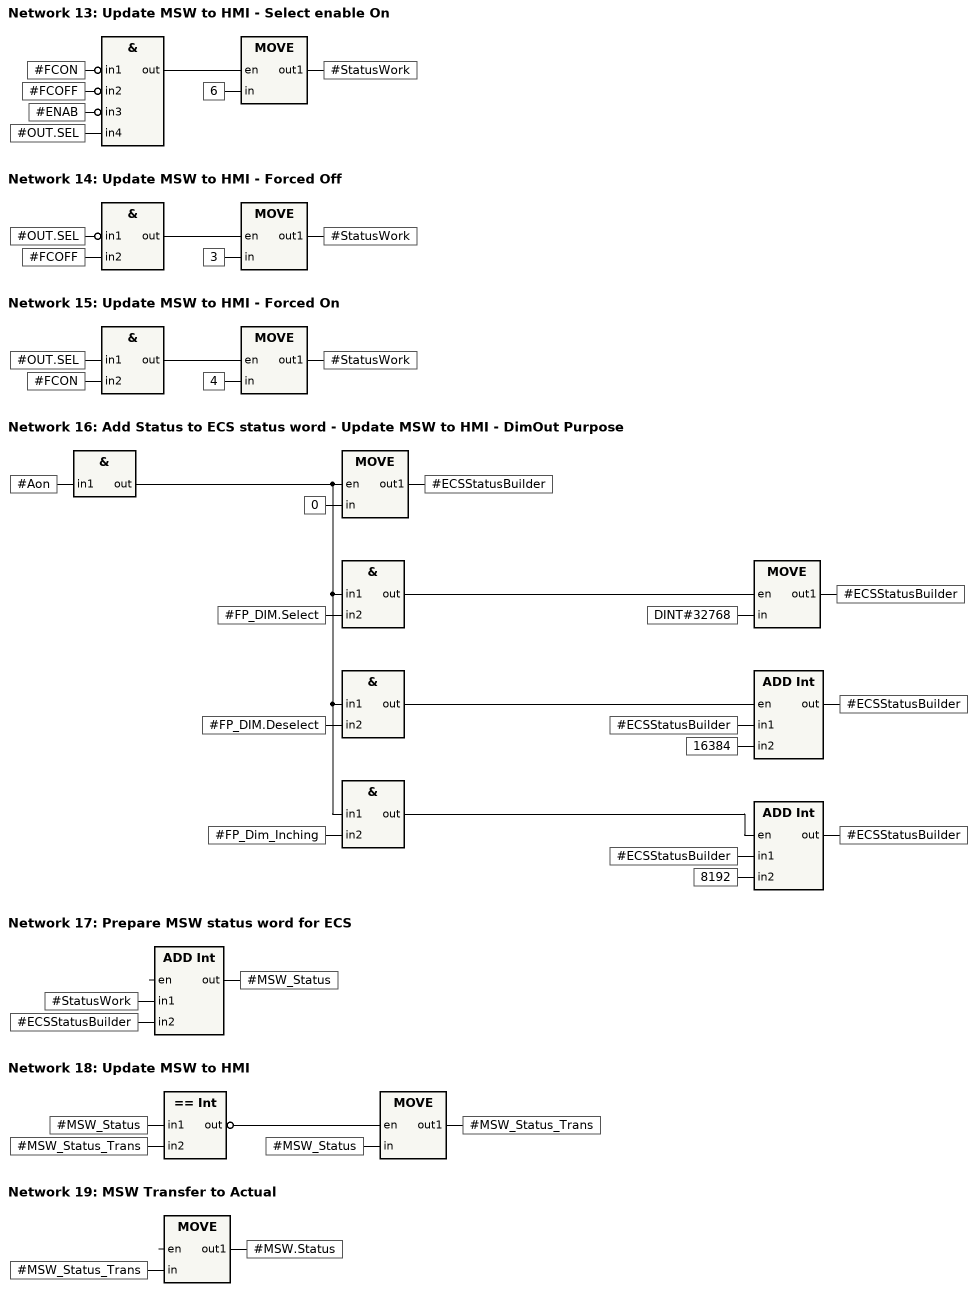
   IF NOT #FCON AND NOT #FCOFF AND NOT #ENAB AND #OUT.SEL THEN #StatusWork := 6; END_IF;
END_REGION

REGION Network 14: Update MSW to HMI - Forced Off
   IF NOT #OUT.SEL AND #FCOFF THEN #StatusWork := 3; END_IF;
END_REGION

REGION Network 15: Update MSW to HMI - Forced On
   IF #OUT.SEL AND #FCON THEN #StatusWork := 4; END_IF;
END_REGION

REGION Network 16: Add Status to ECS status word - Update MSW to HMI - DimOut Purpose
   // Bit 15 = 32768 - Dim_Select
   // Bit 14 = 16384 - Dim_Deselect
   // Bit 13 = 8192  - Dim Inching
   // Bit 12 = 4096 (spare)
   // Bit 11 = 2048 (spare)
   IF #Aon THEN #ECSStatusBuilder := 0; END_IF;
   IF #Aon AND #FP_DIM.Select THEN #ECSStatusBuilder := DINT#32768; END_IF;
   IF #Aon AND #FP_DIM.Deselect THEN #ECSStatusBuilder := #ECSStatusBuilder + 16384; END_IF;
   IF #Aon AND #FP_Dim_Inching THEN #ECSStatusBuilder := #ECSStatusBuilder + 8192; END_IF;
END_REGION

REGION Network 17: Prepare MSW status word for ECS
   #MSW_Status := #StatusWork + #ECSStatusBuilder;
END_REGION

REGION Network 18: Update MSW to HMI
   IF NOT (#MSW_Status = #MSW_Status_Trans) THEN #MSW_Status_Trans := #MSW_Status; END_IF;
END_REGION

REGION Network 19: MSW Transfer to Actual
   #MSW.Status := #MSW_Status_Trans;
END_REGION

REGION Network 20: Write STAT to OUT
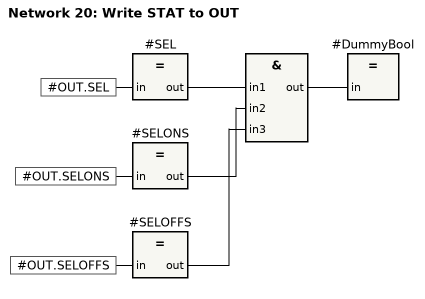
   #SEL := #OUT.SEL;
   #SELONS := #OUT.SELONS;
   #SELOFFS := #OUT.SELOFFS;
   #DummyBool := #OUT.SEL AND #OUT.SELONS AND #OUT.SELOFFS;
END_REGION
END_FUNCTION_BLOCK

FUNCTION_BLOCK "ACESYS_TOTALIZER"   // FB206, FBD
TITLE = ACESYS V8.0 - Build 002 - TOTALIZER
{ S7_Optimized_Access := 'FALSE' }
AUTHOR : FLSmidth
FAMILY : ACESYS
NAME : TOTALIZE
VERSION : 8.0
   VAR_INPUT
      CNT_EN : Bool;   // Counting Enable
      CNT : Bool;   // Counter Pulse
      RESET : Bool;   // Reset Counter Value
      DI_AI : Bool;   // Select Sum. Pulses or Analog-val ("0" = Dig./"1"=Ana.)
      AI : Real;   // Analog Value (Eng. Units)
   END_VAR
   VAR_OUTPUT
      COUNT : Real;   // Actual Counter Value
      Tot_Hour : Real;   // Tot. Totalizer, Base Hour
      Tot_Day : Real;   // Tot. Totalizer, Base Day
      Tot_Month : Real;
      Tot_Year : Real;   // Tot. Totalizer, Base Year
      MSW : DInt;
   END_VAR
   VAR_IN_OUT
      Token : "ACESYS_TOKEN";
   END_VAR
   VAR
      BlockInfo : Struct
         Ace_Version : Int;   // Acesys Block Version Number
         Ace_BuildNo : Int;   // Acesys Block Build Number
         State_Act : Int;   // Actual State Number
         State_Prev : Int;   // Previous State Number
         DB_Number : Int;   // Block Instance DB Number
      END_STRUCT;
      FP_CMD : Struct   // Faceplate Commands
         Spare_08 : Bool;
         Spare_09 : Bool;
         Spare_10 : Bool;
         Spare_11 : Bool;
         Spare_12 : Bool;
         Spare_13 : Bool;
         Spare_14 : Bool;
         AckAlarm : Bool;
         Reset : Bool;
         Spare_01 : Bool;
         Spare_02 : Bool;
         Spare_03 : Bool;
         Spare_04 : Bool;
         Spare_05 : Bool;
         Spare_06 : Bool;
         Spare_07 : Bool;
      END_STRUCT;
      FP_EN : Struct
         Reset : Bool;
      END_STRUCT;
      FP_SEL : Struct
         AI_Type_1 : Bool;   // Analog Value x/s
         AI_Type_2 : Bool;   // Analog Value x/min
         AI_Type_3 : Bool;   // Analog Value x/h
         COUNT_Factor_1 : Bool;   // AI / COUNT Ratio : 1:1
         COUNT_Factor_2 : Bool;   // AI / COUNT Ratio : 10:1
         COUNT_Factor_3 : Bool;   // AI / COUNT Ratio : 100:1
         COUNT_Factor_4 : Bool;   // AI / COUNT Ratio : 1000:1
         User_Hour : Bool;
         User_Day : Bool;
         User_Month : Bool;
         User_Year : Bool;
         User_Defined : Bool;
      END_STRUCT;
      FP_PAR : Struct
         Prev_Hour : Real;   // Save Old Counter register
         Prev_Day : Real;   // Save Old Counter register
         Prev_Month : Real;   // Save Old Counter register
         Prev_Year : Real;   // Save Old Counter register
         Prev_User : Real;   // Save Old Counter registe
      END_STRUCT;
      FP_DIM : Struct
         Reset : Bool;
      END_STRUCT;
      FP_SHOW : Struct
         Reset : Bool;
      END_STRUCT;
      ONS : Struct
         AI_Type_1 : Bool;
         AI_Type_2 : Bool;
         AI_Type_3 : Bool;
         COUNT_Factor_1 : Bool;
         COUNT_Factor_2 : Bool;
         COUNT_Factor_3 : Bool;
         COUNT_Factor_4 : Bool;
         User_Hour : Bool;
         User_Day : Bool;
         User_Month : Bool;
         User_Year : Bool;
         User_Defined : Bool;
         CNT : Bool;
         Reset : Bool;
         SecPulse1 : Bool;
         SecPulse2 : Bool;
      END_STRUCT;
      CMD_Reset : Bool;   // Reset Counters
      Sec_Pulse : Bool;
      Spare6 : Bool;
      Spare5 : Bool;
      Spare4 : Bool;
      Spare3 : Bool;
      Spare2 : Bool;
      Spare1 : Bool;
      inc_tmr_Real : LReal;   // Time elapsed since last block call (ms)
      IncrementVal : LReal;
      Selected_Factor : LReal;   // Ratio x:1
      Hour_Int : LReal;
      Day_Int : LReal;
      Month_Int : LReal;
      Year_Int : LReal;
      User_int : LReal;
      AI_Cal_Lreal : LReal;
      Runtime_RetVal : LReal;
      Runtime_Result : LReal;
      Runtime_Mem1 : LReal;
   END_VAR
   VAR_TEMP
      Aon : Bool;
      Aoff : Bool;
      DummyBool : Bool;
      DummyReal : Real;
      DummyLReal : LReal;
      DummyDint : DInt;
      AI_Cal : Real;
      DummyDword : DWord;
   END_VAR
   VAR_TEMP   // added for the SCL form of the ladder/FBD networks
      _w1 : Bool;
      _w2 : Bool;
   END_VAR
BEGIN

REGION Network 1
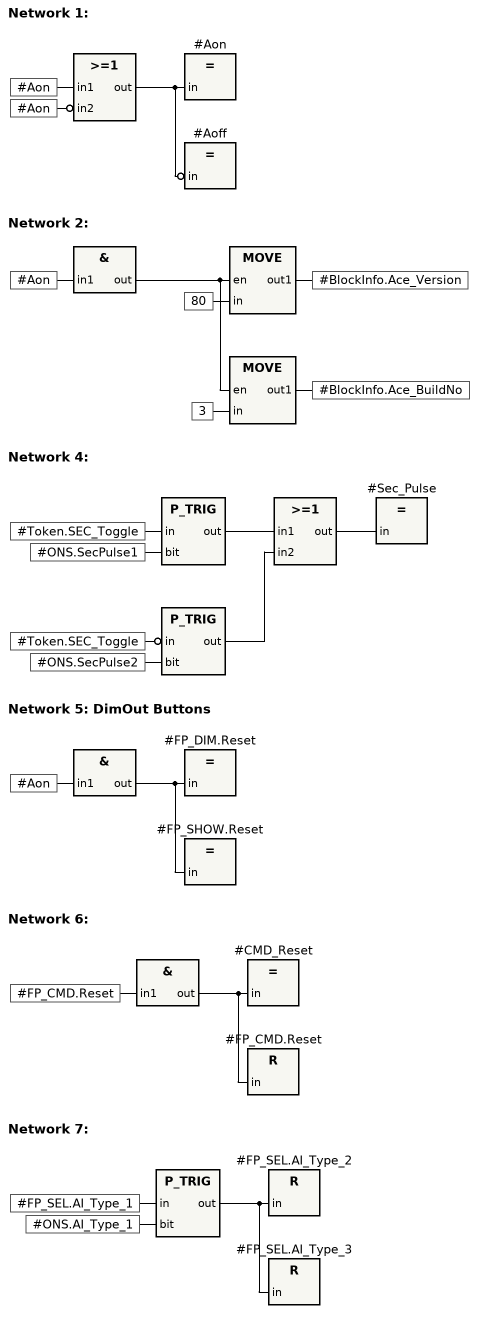
   #Aon := #Aon OR NOT #Aon;
   #Aoff := NOT #Aon;
END_REGION

REGION Network 2
   // Build 003 - Nw26 Runtime_Result replaced in Multiplication Input
   IF #Aon THEN
       #BlockInfo.Ace_Version := 80;
       #BlockInfo.Ace_BuildNo := 3;
   END_IF;
END_REGION

REGION Network 3 (STL): Instance DB Number to Faceplate
         L     DINO;
         T     #BlockInfo.DB_Number;
END_REGION

REGION Network 4
   #_w1 := #Token.SEC_Toggle AND NOT #ONS.SecPulse1;   // rising edge
   #ONS.SecPulse1 := #Token.SEC_Toggle;
   #_w2 := NOT #Token.SEC_Toggle AND NOT #ONS.SecPulse2;   // rising edge
   #ONS.SecPulse2 := NOT #Token.SEC_Toggle;
   #Sec_Pulse := #_w1 OR #_w2;
END_REGION

REGION Network 5: DimOut Buttons
   #FP_DIM.Reset := #Aon;
   #FP_SHOW.Reset := #Aon;
END_REGION

REGION Network 6
   // >>>>>Automatic Dep_CMD when use of block interface<<<<<<
   #CMD_Reset := #FP_CMD.Reset;
   IF #FP_CMD.Reset THEN #FP_CMD.Reset := FALSE; END_IF;
END_REGION

REGION Network 7
   // >>>>>Select Time Base for Input Engineering Value<<<<<<
   // (sec, minute, hour)
   #_w1 := #FP_SEL.AI_Type_1 AND NOT #ONS.AI_Type_1;   // rising edge
   #ONS.AI_Type_1 := #FP_SEL.AI_Type_1;
   IF #_w1 THEN
       #FP_SEL.AI_Type_2 := FALSE;
       #FP_SEL.AI_Type_3 := FALSE;
   END_IF;
END_REGION

REGION Network 8
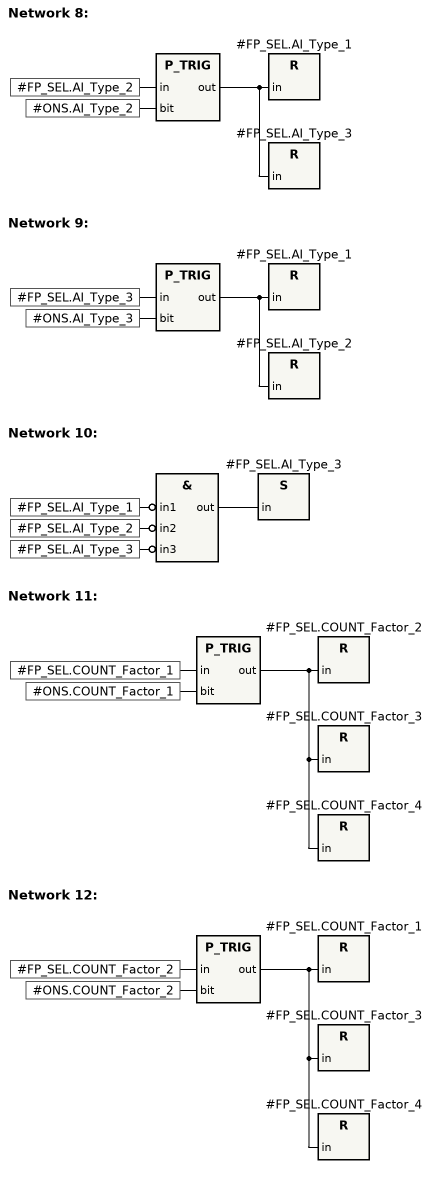
   #_w1 := #FP_SEL.AI_Type_2 AND NOT #ONS.AI_Type_2;   // rising edge
   #ONS.AI_Type_2 := #FP_SEL.AI_Type_2;
   IF #_w1 THEN
       #FP_SEL.AI_Type_1 := FALSE;
       #FP_SEL.AI_Type_3 := FALSE;
   END_IF;
END_REGION

REGION Network 9
   #_w1 := #FP_SEL.AI_Type_3 AND NOT #ONS.AI_Type_3;   // rising edge
   #ONS.AI_Type_3 := #FP_SEL.AI_Type_3;
   IF #_w1 THEN
       #FP_SEL.AI_Type_1 := FALSE;
       #FP_SEL.AI_Type_2 := FALSE;
   END_IF;
END_REGION

REGION Network 10
   IF NOT #FP_SEL.AI_Type_1 AND NOT #FP_SEL.AI_Type_2 AND NOT #FP_SEL.AI_Type_3 THEN
       #FP_SEL.AI_Type_3 := TRUE;
   END_IF;
END_REGION

REGION Network 11
   // >>>>>Select Factor<<<<<
   // (Ratio 1:1, 10:1, 100:1, 1000:1)
   #_w1 := #FP_SEL.COUNT_Factor_1 AND NOT #ONS.COUNT_Factor_1;   // rising edge
   #ONS.COUNT_Factor_1 := #FP_SEL.COUNT_Factor_1;
   IF #_w1 THEN
       #FP_SEL.COUNT_Factor_2 := FALSE;
       #FP_SEL.COUNT_Factor_3 := FALSE;
       #FP_SEL.COUNT_Factor_4 := FALSE;
   END_IF;
END_REGION

REGION Network 12
   #_w1 := #FP_SEL.COUNT_Factor_2 AND NOT #ONS.COUNT_Factor_2;   // rising edge
   #ONS.COUNT_Factor_2 := #FP_SEL.COUNT_Factor_2;
   IF #_w1 THEN
       #FP_SEL.COUNT_Factor_1 := FALSE;
       #FP_SEL.COUNT_Factor_3 := FALSE;
       #FP_SEL.COUNT_Factor_4 := FALSE;
   END_IF;
END_REGION

REGION Network 13
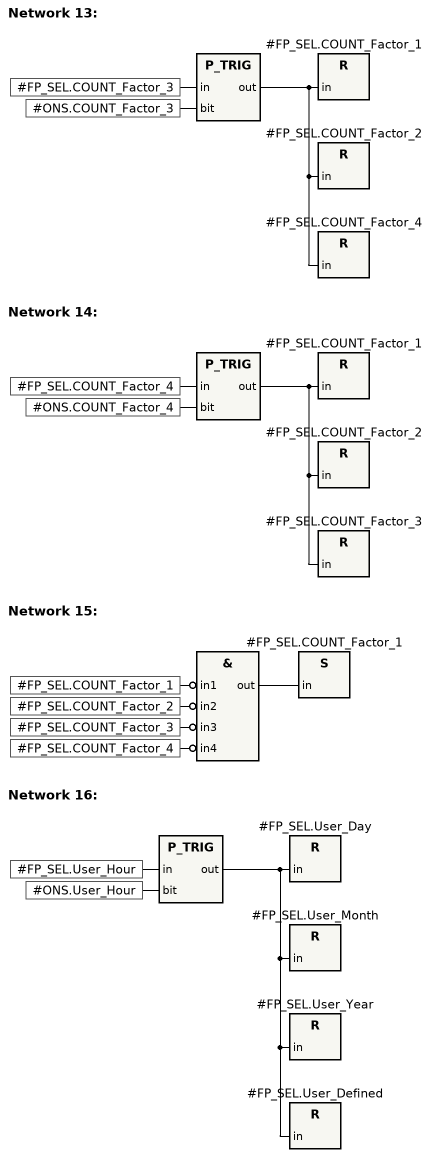
   #_w1 := #FP_SEL.COUNT_Factor_3 AND NOT #ONS.COUNT_Factor_3;   // rising edge
   #ONS.COUNT_Factor_3 := #FP_SEL.COUNT_Factor_3;
   IF #_w1 THEN
       #FP_SEL.COUNT_Factor_1 := FALSE;
       #FP_SEL.COUNT_Factor_2 := FALSE;
       #FP_SEL.COUNT_Factor_4 := FALSE;
   END_IF;
END_REGION

REGION Network 14
   #_w1 := #FP_SEL.COUNT_Factor_4 AND NOT #ONS.COUNT_Factor_4;   // rising edge
   #ONS.COUNT_Factor_4 := #FP_SEL.COUNT_Factor_4;
   IF #_w1 THEN
       #FP_SEL.COUNT_Factor_1 := FALSE;
       #FP_SEL.COUNT_Factor_2 := FALSE;
       #FP_SEL.COUNT_Factor_3 := FALSE;
   END_IF;
END_REGION

REGION Network 15
   IF NOT #FP_SEL.COUNT_Factor_1 AND NOT #FP_SEL.COUNT_Factor_2 AND NOT #FP_SEL.COUNT_Factor_3 AND NOT #FP_SEL.COUNT_Factor_4 THEN
       #FP_SEL.COUNT_Factor_1 := TRUE;
   END_IF;
END_REGION

REGION Network 16
   // >>>>>Select User Defined value to Output and  MSW<<<<<
   #_w1 := #FP_SEL.User_Hour AND NOT #ONS.User_Hour;   // rising edge
   #ONS.User_Hour := #FP_SEL.User_Hour;
   IF #_w1 THEN
       #FP_SEL.User_Day := FALSE;
       #FP_SEL.User_Month := FALSE;
       #FP_SEL.User_Year := FALSE;
       #FP_SEL.User_Defined := FALSE;
   END_IF;
END_REGION

REGION Network 17
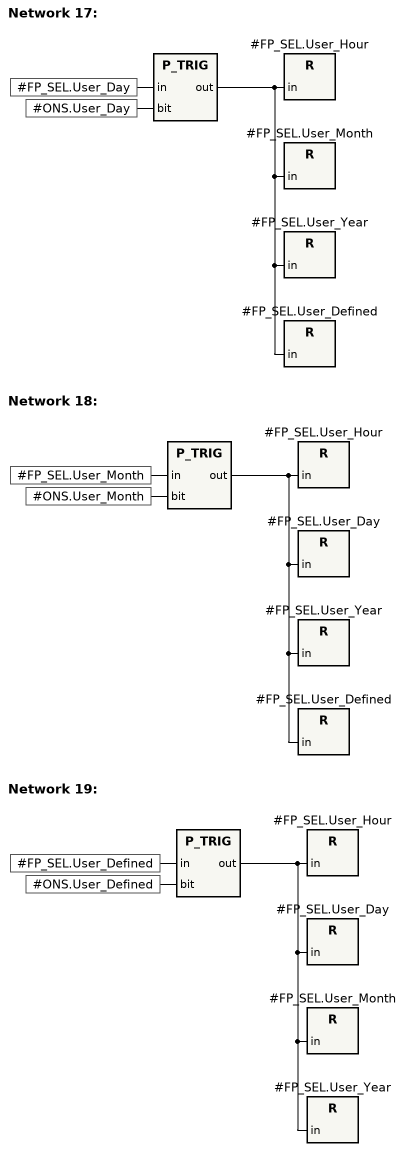
   #_w1 := #FP_SEL.User_Day AND NOT #ONS.User_Day;   // rising edge
   #ONS.User_Day := #FP_SEL.User_Day;
   IF #_w1 THEN
       #FP_SEL.User_Hour := FALSE;
       #FP_SEL.User_Month := FALSE;
       #FP_SEL.User_Year := FALSE;
       #FP_SEL.User_Defined := FALSE;
   END_IF;
END_REGION

REGION Network 18
   #_w1 := #FP_SEL.User_Month AND NOT #ONS.User_Month;   // rising edge
   #ONS.User_Month := #FP_SEL.User_Month;
   IF #_w1 THEN
       #FP_SEL.User_Hour := FALSE;
       #FP_SEL.User_Day := FALSE;
       #FP_SEL.User_Year := FALSE;
       #FP_SEL.User_Defined := FALSE;
   END_IF;
END_REGION

REGION Network 19
   #_w1 := #FP_SEL.User_Defined AND NOT #ONS.User_Defined;   // rising edge
   #ONS.User_Defined := #FP_SEL.User_Defined;
   IF #_w1 THEN
       #FP_SEL.User_Hour := FALSE;
       #FP_SEL.User_Day := FALSE;
       #FP_SEL.User_Month := FALSE;
       #FP_SEL.User_Year := FALSE;
   END_IF;
END_REGION

REGION Network 20
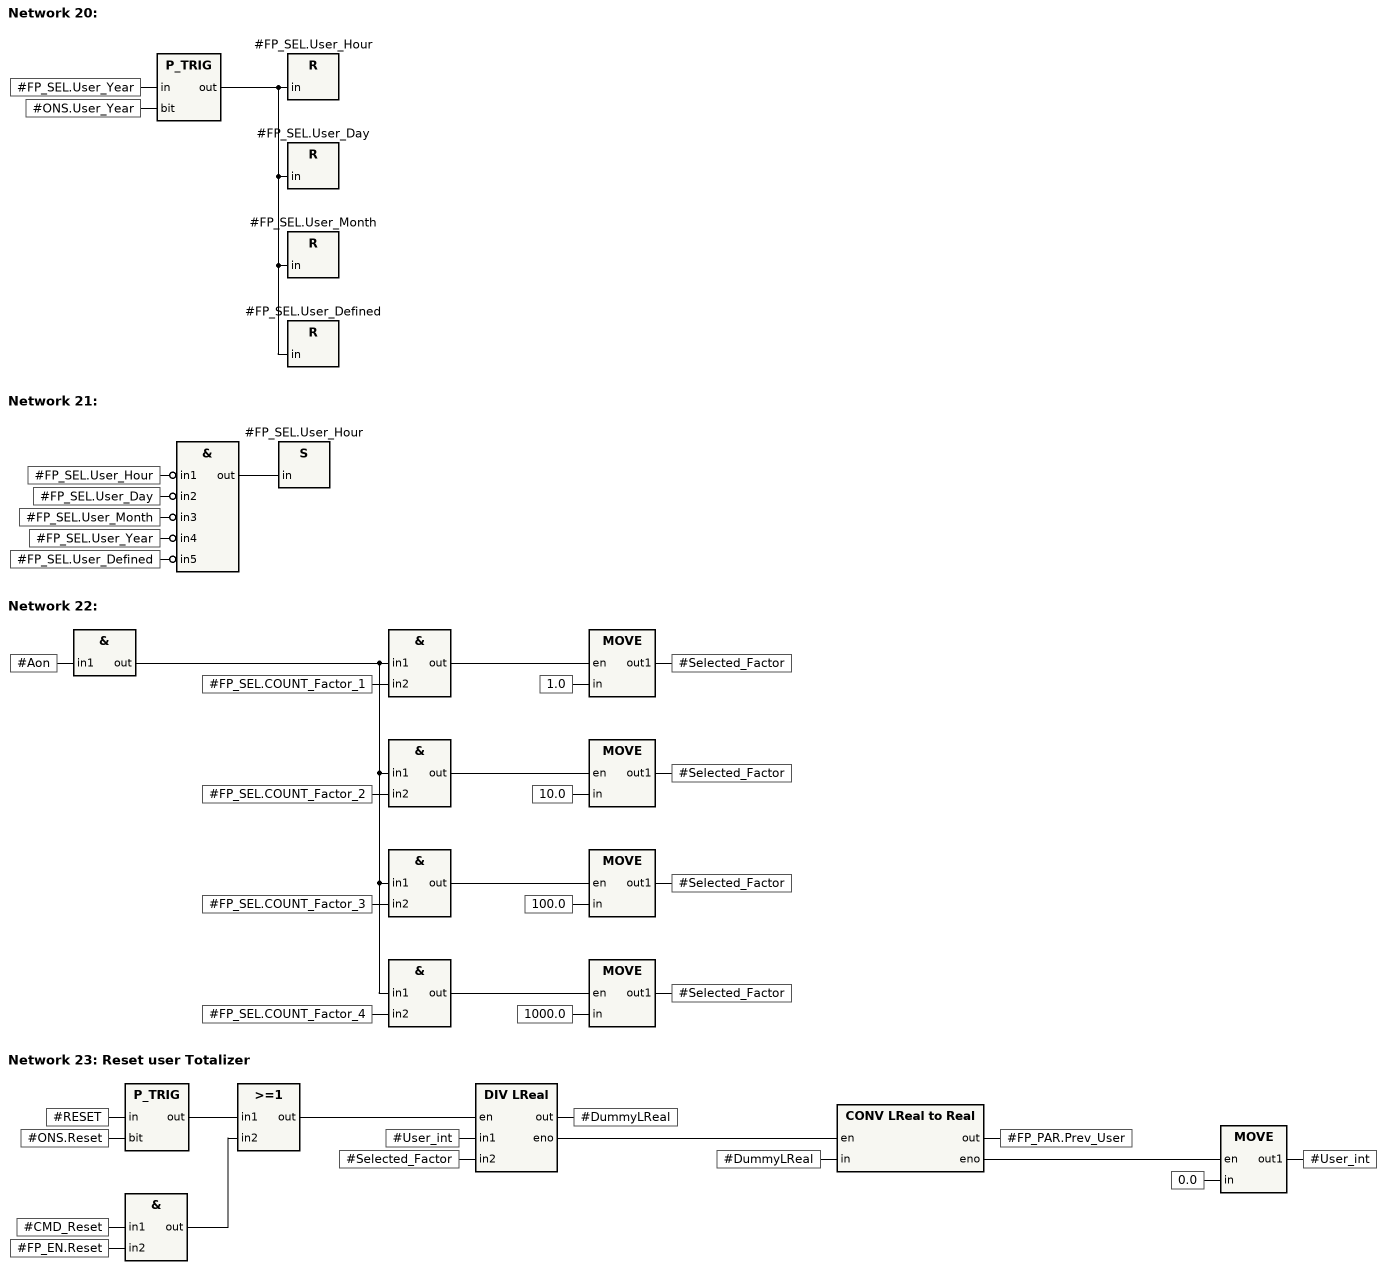
   #_w1 := #FP_SEL.User_Year AND NOT #ONS.User_Year;   // rising edge
   #ONS.User_Year := #FP_SEL.User_Year;
   IF #_w1 THEN
       #FP_SEL.User_Hour := FALSE;
       #FP_SEL.User_Day := FALSE;
       #FP_SEL.User_Month := FALSE;
       #FP_SEL.User_Defined := FALSE;
   END_IF;
END_REGION

REGION Network 21
   IF NOT #FP_SEL.User_Hour AND NOT #FP_SEL.User_Day AND NOT #FP_SEL.User_Month AND NOT #FP_SEL.User_Year AND NOT #FP_SEL.User_Defined THEN
       #FP_SEL.User_Hour := TRUE;
   END_IF;
END_REGION

REGION Network 22
   // >>>>>Get Selected Factor<<<<<
   IF #Aon AND #FP_SEL.COUNT_Factor_1 THEN #Selected_Factor := 1.0; END_IF;
   IF #Aon AND #FP_SEL.COUNT_Factor_2 THEN #Selected_Factor := 10.0; END_IF;
   IF #Aon AND #FP_SEL.COUNT_Factor_3 THEN #Selected_Factor := 100.0; END_IF;
   IF #Aon AND #FP_SEL.COUNT_Factor_4 THEN #Selected_Factor := 1000.0; END_IF;
END_REGION

REGION Network 23: Reset user Totalizer
   // Build 002 - 01.Feb.2016 : Factor is in included before the value is send to 
   // Prev_User
   // ENO of a box is taken as its EN; it also drops when the box reports an error
   #_w1 := #RESET AND NOT #ONS.Reset;   // rising edge
   #ONS.Reset := #RESET;
   IF #_w1 OR (#CMD_Reset AND #FP_EN.Reset) THEN
       #DummyLReal := #User_int / #Selected_Factor;
       #FP_PAR.Prev_User := LREAL_TO_REAL(#DummyLReal);
       #User_int := 0.0;
   END_IF;
END_REGION

REGION Network 24: Reset and Save prev. :Hour, Day, Month, Year
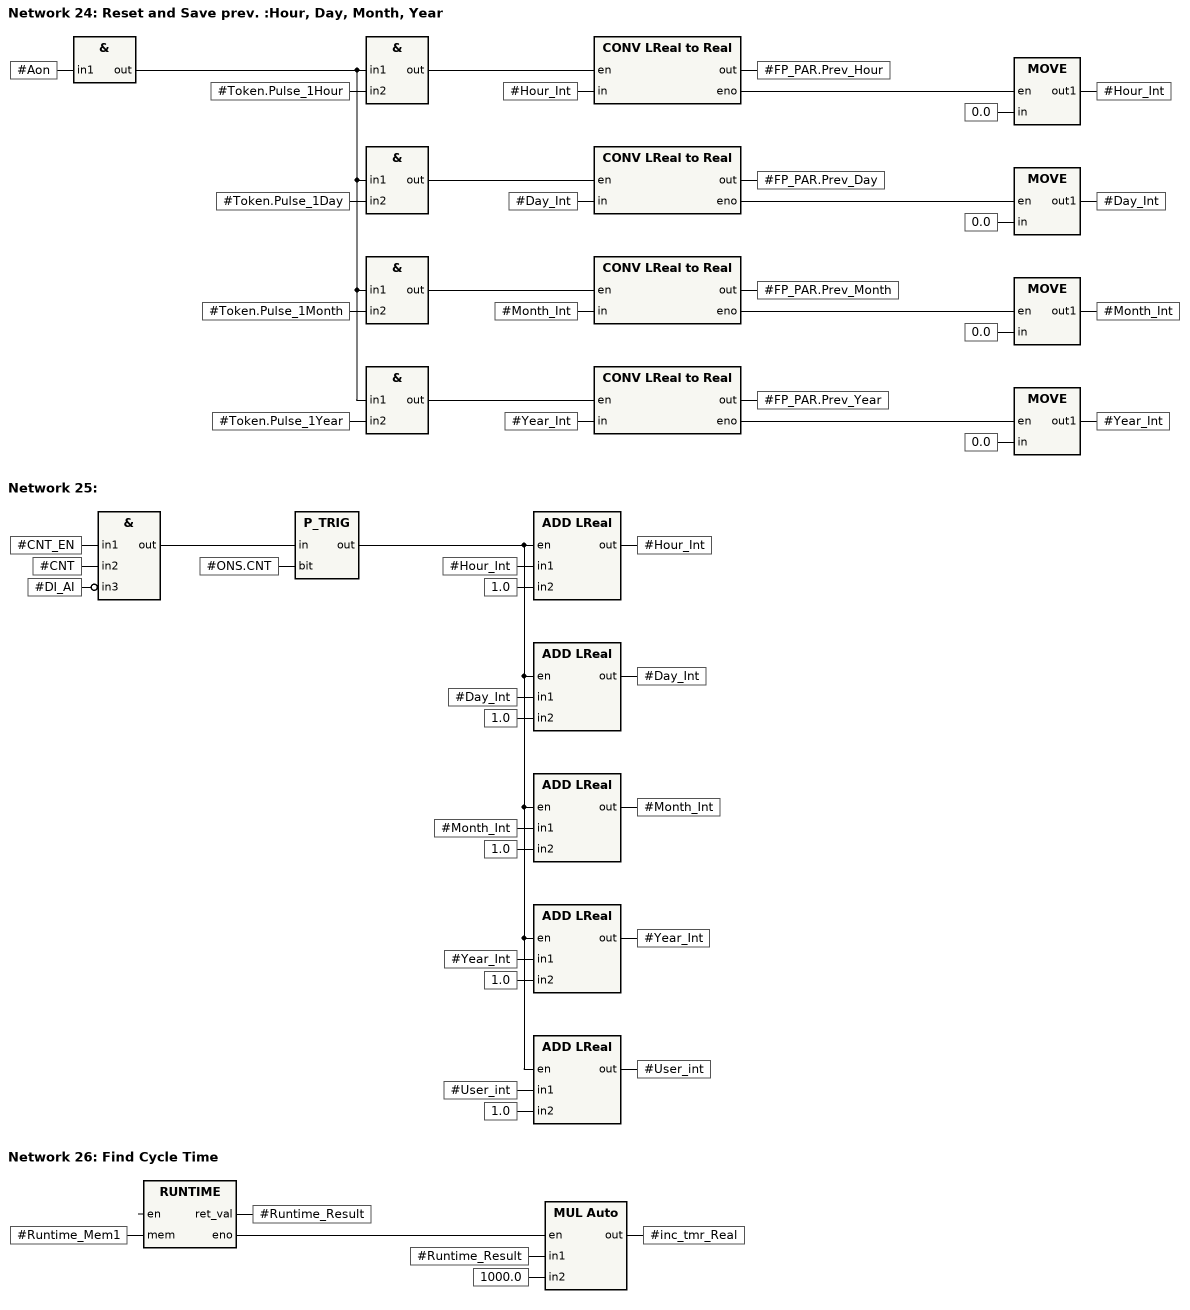
   IF #Aon AND #Token.Pulse_1Hour THEN
       #FP_PAR.Prev_Hour := LREAL_TO_REAL(#Hour_Int);
       #Hour_Int := 0.0;
   END_IF;
   IF #Aon AND #Token.Pulse_1Day THEN
       #FP_PAR.Prev_Day := LREAL_TO_REAL(#Day_Int);
       #Day_Int := 0.0;
   END_IF;
   IF #Aon AND #Token.Pulse_1Month THEN
       #FP_PAR.Prev_Month := LREAL_TO_REAL(#Month_Int);
       #Month_Int := 0.0;
   END_IF;
   IF #Aon AND #Token.Pulse_1Year THEN
       #FP_PAR.Prev_Year := LREAL_TO_REAL(#Year_Int);
       #Year_Int := 0.0;
   END_IF;
END_REGION

REGION Network 25
   // >>>>>Digital Counting<<<<<
   #_w1 := #CNT_EN AND #CNT AND NOT #DI_AI;
   #_w2 := #_w1 AND NOT #ONS.CNT;   // rising edge
   #ONS.CNT := #_w1;
   IF #_w2 THEN
       #Hour_Int := #Hour_Int + 1.0;
       #Day_Int := #Day_Int + 1.0;
       #Month_Int := #Month_Int + 1.0;
       #Year_Int := #Year_Int + 1.0;
       #User_int := #User_int + 1.0;
   END_IF;
END_REGION

REGION Network 26: Find Cycle Time
   // Build 003 - Runtime_Result replaced in Multiplication Input
   // no SCL statement known for Runtime: written as a call
   // ENO of a box is taken as its EN; it also drops when the box reports an error
   #Runtime_Result := Runtime(mem := #Runtime_Mem1);
   #inc_tmr_Real := #Runtime_Result * 1000.0;
END_REGION

REGION Network 27
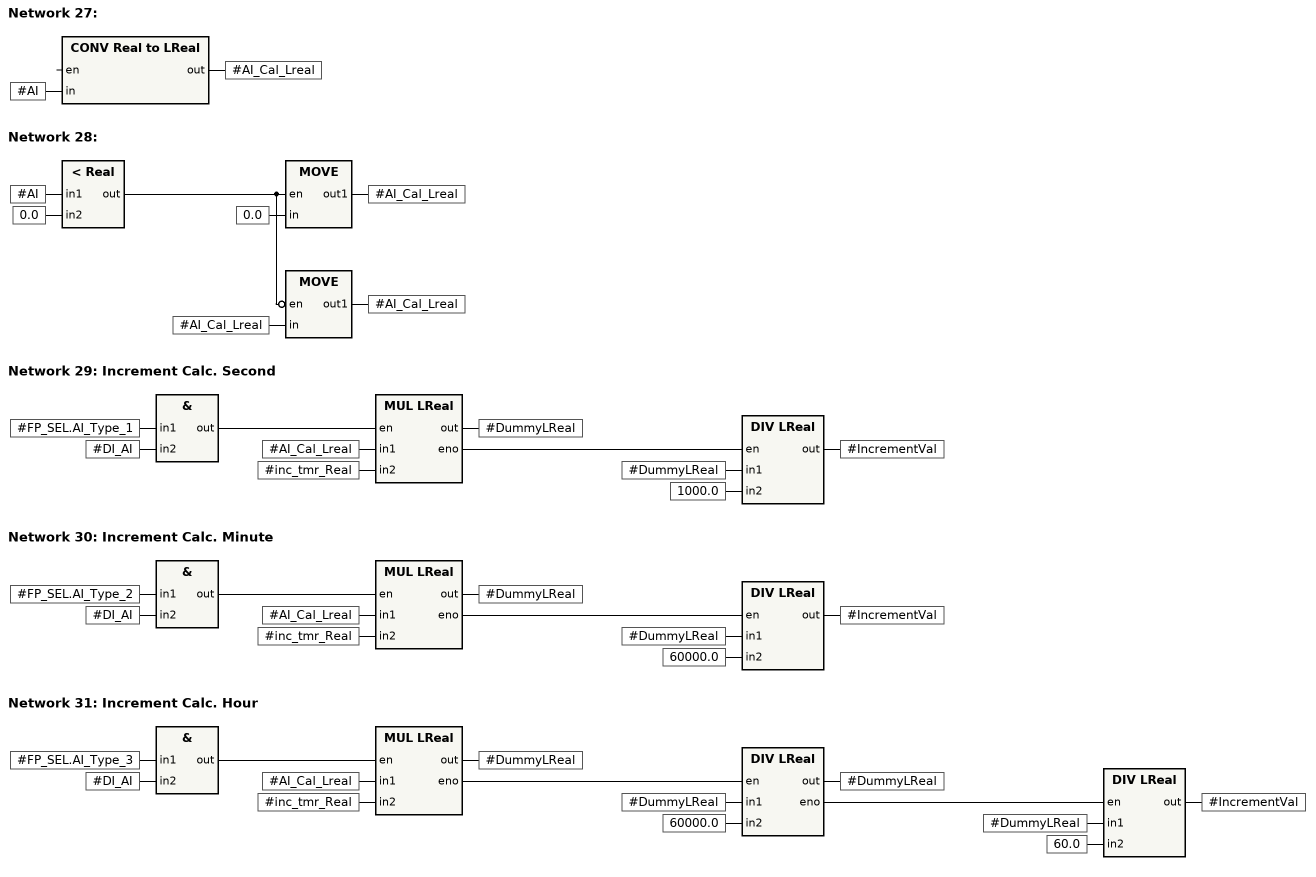
   #AI_Cal_Lreal := REAL_TO_LREAL(#AI);
END_REGION

REGION Network 28
   // Build 002 - 01.Feb.2016 : AI is clamped to "0"
   #_w1 := #AI < 0.0;
   IF #_w1 THEN #AI_Cal_Lreal := 0.0; END_IF;
   IF NOT #_w1 THEN #AI_Cal_Lreal := #AI_Cal_Lreal; END_IF;
END_REGION

REGION Network 29: Increment Calc. Second
   // Build 002 - 01.Feb.2016 : AI replaced with AI_Cal
   // ENO of a box is taken as its EN; it also drops when the box reports an error
   IF #FP_SEL.AI_Type_1 AND #DI_AI THEN
       #DummyLReal := #AI_Cal_Lreal * #inc_tmr_Real;
       #IncrementVal := #DummyLReal / 1000.0;
   END_IF;
END_REGION

REGION Network 30: Increment Calc. Minute
   // Build 002 - 01.Feb.2016 : AI replaced with AI_Cal
   // ENO of a box is taken as its EN; it also drops when the box reports an error
   IF #FP_SEL.AI_Type_2 AND #DI_AI THEN
       #DummyLReal := #AI_Cal_Lreal * #inc_tmr_Real;
       #IncrementVal := #DummyLReal / 60000.0;
   END_IF;
END_REGION

REGION Network 31: Increment Calc. Hour
   // Build 002 - 01.Feb.2016 : AI replaced with AI_Cal
   // ENO of a box is taken as its EN; it also drops when the box reports an error
   IF #FP_SEL.AI_Type_3 AND #DI_AI THEN
       #DummyLReal := #AI_Cal_Lreal * #inc_tmr_Real;
       #DummyLReal := #DummyLReal / 60000.0;
       #IncrementVal := #DummyLReal / 60.0;
   END_IF;
END_REGION

REGION Network 32
   // >>>>>Increment Base on Analog<<<<<
   // TOTAL Totalizer - Count up analog
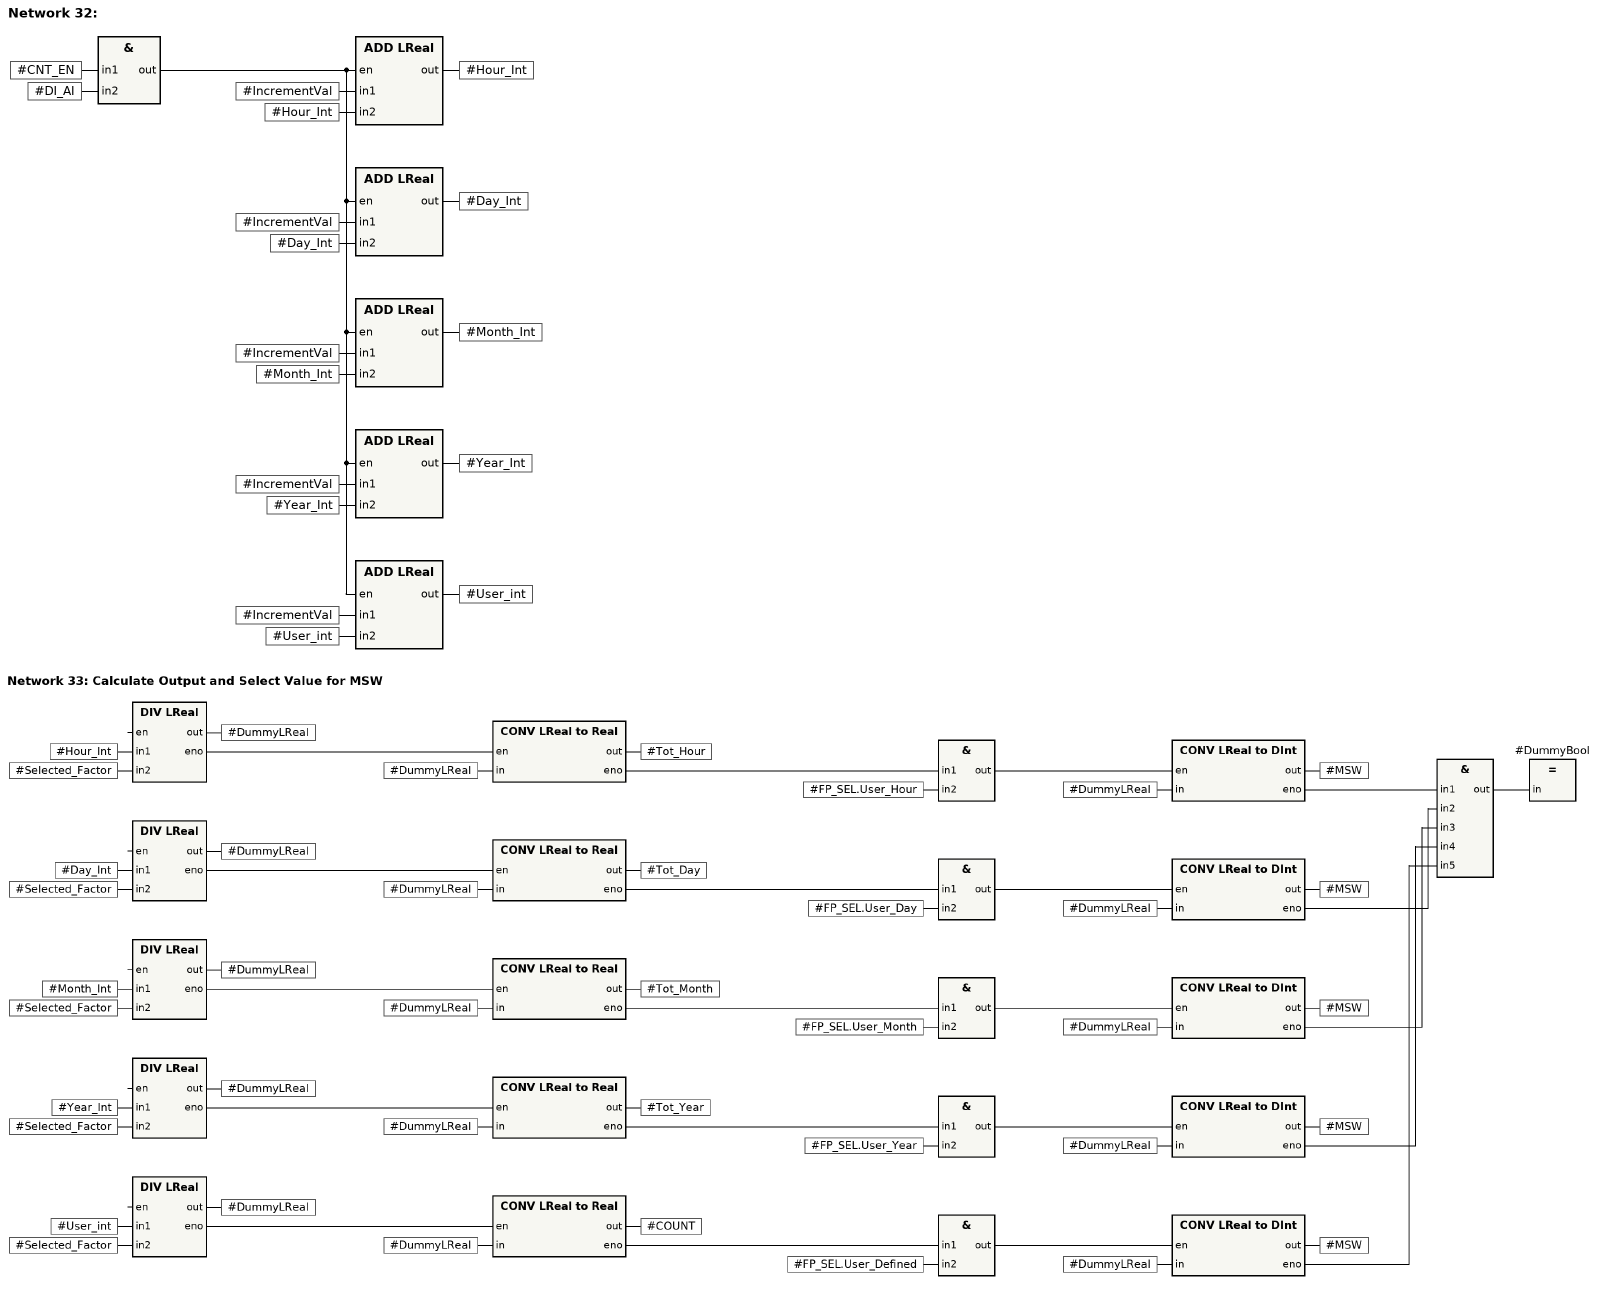
   IF #CNT_EN AND #DI_AI THEN
       #Hour_Int := #IncrementVal + #Hour_Int;
       #Day_Int := #IncrementVal + #Day_Int;
       #Month_Int := #IncrementVal + #Month_Int;
       #Year_Int := #IncrementVal + #Year_Int;
       #User_int := #IncrementVal + #User_int;
   END_IF;
END_REGION

REGION Network 33: Calculate Output and Select Value for MSW
   // ENO of a box is taken as its EN; it also drops when the box reports an error
   #DummyLReal := #Hour_Int / #Selected_Factor;
   #Tot_Hour := LREAL_TO_REAL(#DummyLReal);
   IF #FP_SEL.User_Hour THEN #MSW := LREAL_TO_DINT(#DummyLReal); END_IF;
   #DummyLReal := #Day_Int / #Selected_Factor;
   #Tot_Day := LREAL_TO_REAL(#DummyLReal);
   IF #FP_SEL.User_Day THEN #MSW := LREAL_TO_DINT(#DummyLReal); END_IF;
   #DummyLReal := #Month_Int / #Selected_Factor;
   #Tot_Month := LREAL_TO_REAL(#DummyLReal);
   IF #FP_SEL.User_Month THEN #MSW := LREAL_TO_DINT(#DummyLReal); END_IF;
   #DummyLReal := #Year_Int / #Selected_Factor;
   #Tot_Year := LREAL_TO_REAL(#DummyLReal);
   IF #FP_SEL.User_Year THEN #MSW := LREAL_TO_DINT(#DummyLReal); END_IF;
   #DummyLReal := #User_int / #Selected_Factor;
   #COUNT := LREAL_TO_REAL(#DummyLReal);
   IF #FP_SEL.User_Defined THEN #MSW := LREAL_TO_DINT(#DummyLReal); END_IF;
   #DummyBool := #FP_SEL.User_Hour AND #FP_SEL.User_Day AND #FP_SEL.User_Month AND #FP_SEL.User_Year AND #FP_SEL.User_Defined;
END_REGION
END_FUNCTION_BLOCK

FUNCTION_BLOCK "ACESYS_MD"   // FB207, FBD
TITLE = ACESYS V8.0 - Build 001 - MOTION DETECTOR
{ S7_Optimized_Access := 'FALSE' }
AUTHOR : FLSmidth
FAMILY : ACESYS
NAME : MotionDe
VERSION : 8.0
   VAR_INPUT
      CON : Bool;   // Start Command
      MD : Bool;   // Motion Signal
   END_VAR
   VAR_OUTPUT
      OK : Bool;   // Alarm Status OK
      MSW : "ACESYS_HMI_STAT_32T";
   END_VAR
   VAR_IN_OUT
      TOKEN : "ACESYS_TOKEN";
   END_VAR
   VAR
      BlockInfo : Struct
         Ace_Version : Int;   // Acesys Block Version Number
         Ace_BuildNo : Int;   // Acesys Block Build Number
         State_Act : Int;   // Actual State Number
         State_Prev : Int;   // Previous State Number
         DB_Number : Int;   // Block Instance DB Number
      END_STRUCT;
      FP_CMD : Struct   // Faceplate Commands
         Spare_08 : Bool;
         Spare_09 : Bool;
         Spare_10 : Bool;
         Spare_11 : Bool;
         Spare_12 : Bool;
         Spare_13 : Bool;
         Spare_14 : Bool;
         AckAlarm : Bool;
         Spare_00 : Bool;
         Spare_01 : Bool;
         Spare_02 : Bool;
         Spare_03 : Bool;
         Spare_04 : Bool;
         Spare_05 : Bool;
         Spare_06 : Bool;
         Spare_07 : Bool;
      END_STRUCT;
      FP_SEL : Struct
         MD_Maintain : Bool;
         MD_OnOff : Bool;
         MD_Puls : Bool;
         Keep_Status : Bool;
         MD_TimeBased : Bool;
      END_STRUCT;
      FP_PARM : Struct
         SpeedMonOffDelay_Acc : Int;
         SpeedMonOffDelay_Pre : Int;
         SpeedMonOnDelay_Acc : Int;
         SpeedMonOnDelay_Pre : Int;
         SpeedMonTrigDelay_Acc : Int;
         SpeedMonTrigDelay_Pre : Int;
         MD_Freq_SP : Int;
         MD_Freq_PV : Int;
         TimeBaseMonTime_Acc : Int;
         TimeBaseMonTime_Pre : Int;
         SpeedMonTimeBaseCNT_Acc : Int;
         SpeedMonTimeBaseCNT_Pre : Int;
      END_STRUCT;
      FP_EN : Struct
         ParentSupress : Bool;
      END_STRUCT;
      FP_SIM : "ACESYS_SIM_MD";
      ONS : Struct
         SecPulse1 : Bool;
         SecPulse2 : Bool;
         Acknowledge : Bool;
         MD_Pulse : Bool;
         MD_Maintain : Bool;
         MD_Type_OnOff : Bool;
         MD_Type_Pulse : Bool;
         MD_Type_TimeBased : Bool;
      END_STRUCT;
      StatusWork : Int;
      AlarmNo : Int;
      AlarmNo_Old : Int;
      Sec_Pulse : Bool;   // Pulse Every Second
      CMD_Acknowledge : Bool;
      ALARM_SuppresionActiv : Bool;
      ALARM_SuppresionActiv_1 : Bool;
      ALARM_AlarmPresent : Bool;
      ALARM_WarnPresent : Bool;
      ALARM_Failure_Ack_Requ : Bool;
      ALARM_Warn_Ack_Required : Bool;
      SpeedMonOnDelay_Done : Bool;
      SpeedMonOffDelay_Done : Bool;
      SpeedMonTrigDelay_Done : Bool;
      MD_Pulse : Bool;
      Keep_MD_Alarm : Bool;
      TimeBase_Done : Bool;
      TimeBase_TrigAlarm : Bool;
      SpeedMonOnDelay_Mem : Int;
      SpeedMonOffDelay_Mem : Int;
      SpeedMonTrigDelay_Mem : Int;
      TimeBaseMonTime_Mem : Int;
      MD_Time : DInt;
      MD_Time_DINT : DInt;
      MD_Timer : TON_TIME;
      OUT : Struct
         OK : Bool;
         MSW_EXT_ALARMFAILUNACK : Bool;
      END_STRUCT;
      MSW_Status_Trans : Int;
   END_VAR
   VAR_TEMP
      Aon : Bool;
      Aoff : Bool;
      DummyBool : Bool;
      DummyDInt : DInt;
   END_VAR
   VAR_TEMP   // added for the SCL form of the ladder/FBD networks
      _w1 : Bool;
      _w2 : Bool;
   END_VAR
BEGIN

REGION Network 1: Always On
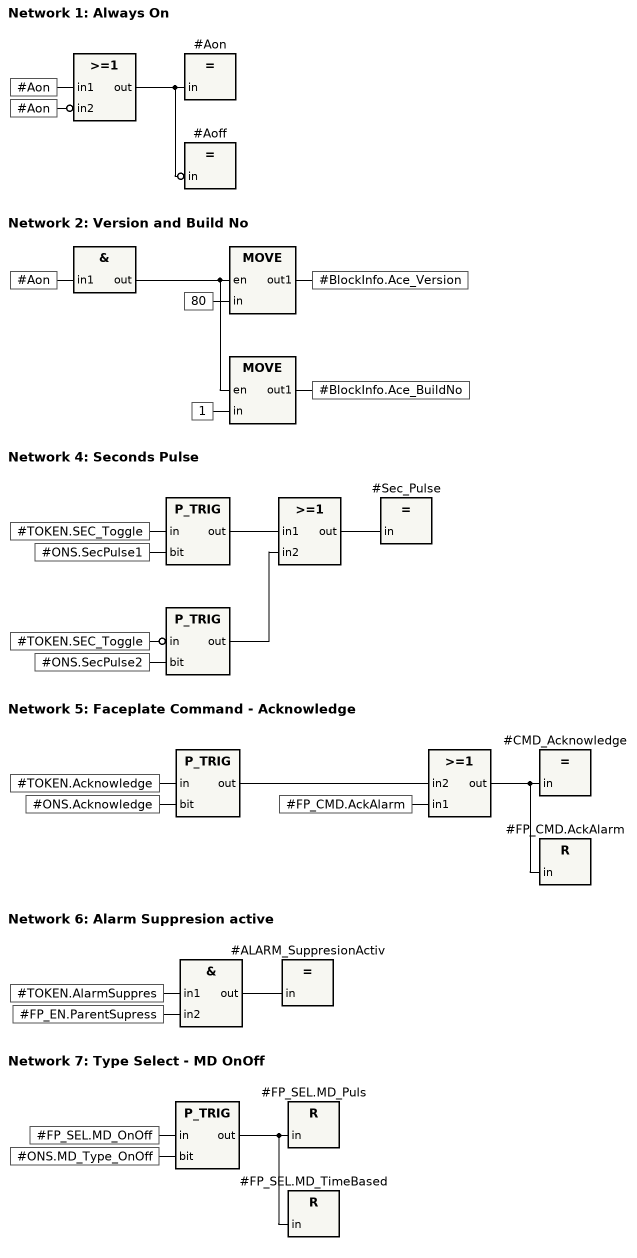
   #Aon := #Aon OR NOT #Aon;
   #Aoff := NOT #Aon;
END_REGION

REGION Network 2: Version and Build No
   IF #Aon THEN
       #BlockInfo.Ace_Version := 80;
       #BlockInfo.Ace_BuildNo := 1;
   END_IF;
END_REGION

REGION Network 3 (STL): Instance DB Number to Faceplate
         L     DINO;
         T     #BlockInfo.DB_Number;
END_REGION

REGION Network 4: Seconds Pulse
   #_w1 := #TOKEN.SEC_Toggle AND NOT #ONS.SecPulse1;   // rising edge
   #ONS.SecPulse1 := #TOKEN.SEC_Toggle;
   #_w2 := NOT #TOKEN.SEC_Toggle AND NOT #ONS.SecPulse2;   // rising edge
   #ONS.SecPulse2 := NOT #TOKEN.SEC_Toggle;
   #Sec_Pulse := #_w1 OR #_w2;
END_REGION

REGION Network 5: Faceplate Command - Acknowledge
   #_w1 := #TOKEN.Acknowledge AND NOT #ONS.Acknowledge;   // rising edge
   #ONS.Acknowledge := #TOKEN.Acknowledge;
   #CMD_Acknowledge := #_w1 OR #FP_CMD.AckAlarm;
   IF #CMD_Acknowledge THEN #FP_CMD.AckAlarm := FALSE; END_IF;
END_REGION

REGION Network 6: Alarm Suppresion active
   #ALARM_SuppresionActiv := #TOKEN.AlarmSuppres AND #FP_EN.ParentSupress;
END_REGION

REGION Network 7: Type Select - MD OnOff
   #_w1 := #FP_SEL.MD_OnOff AND NOT #ONS.MD_Type_OnOff;   // rising edge
   #ONS.MD_Type_OnOff := #FP_SEL.MD_OnOff;
   IF #_w1 THEN
       #FP_SEL.MD_Puls := FALSE;
       #FP_SEL.MD_TimeBased := FALSE;
   END_IF;
END_REGION

REGION Network 8: Type Select - MD Pulse
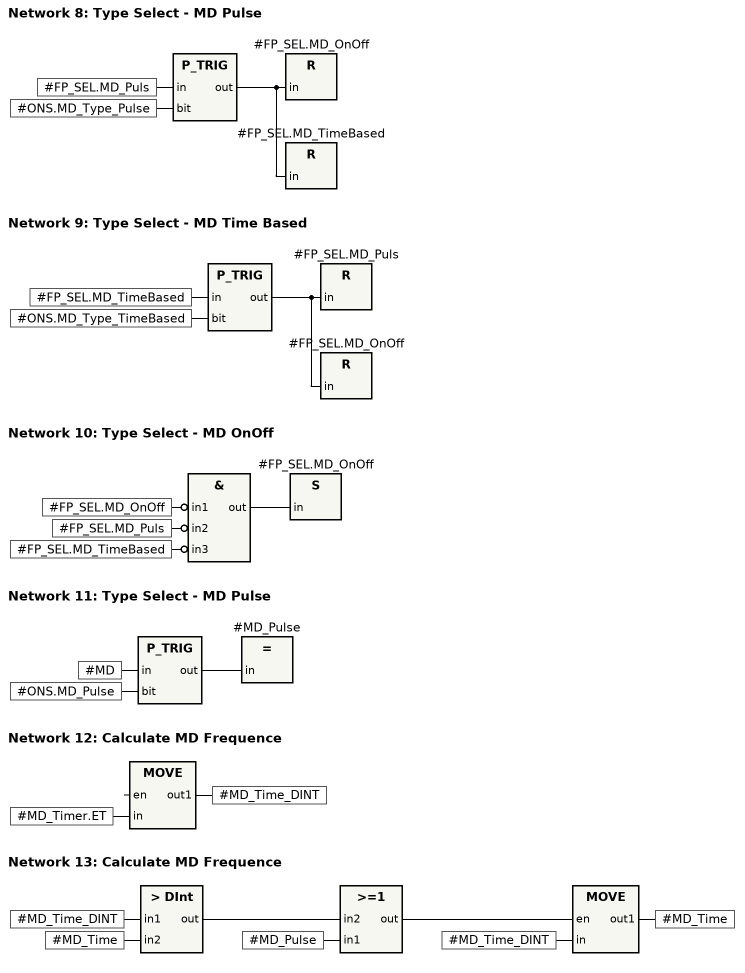
   #_w1 := #FP_SEL.MD_Puls AND NOT #ONS.MD_Type_Pulse;   // rising edge
   #ONS.MD_Type_Pulse := #FP_SEL.MD_Puls;
   IF #_w1 THEN
       #FP_SEL.MD_OnOff := FALSE;
       #FP_SEL.MD_TimeBased := FALSE;
   END_IF;
END_REGION

REGION Network 9: Type Select - MD Time Based
   #_w1 := #FP_SEL.MD_TimeBased AND NOT #ONS.MD_Type_TimeBased;   // rising edge
   #ONS.MD_Type_TimeBased := #FP_SEL.MD_TimeBased;
   IF #_w1 THEN
       #FP_SEL.MD_Puls := FALSE;
       #FP_SEL.MD_OnOff := FALSE;
   END_IF;
END_REGION

REGION Network 10: Type Select - MD OnOff
   IF NOT #FP_SEL.MD_OnOff AND NOT #FP_SEL.MD_Puls AND NOT #FP_SEL.MD_TimeBased THEN
       #FP_SEL.MD_OnOff := TRUE;
   END_IF;
END_REGION

REGION Network 11: Type Select - MD Pulse
   #_w1 := #MD AND NOT #ONS.MD_Pulse;   // rising edge
   #ONS.MD_Pulse := #MD;
   #MD_Pulse := #_w1;
END_REGION

REGION Network 12: Calculate MD Frequence
   #MD_Time_DINT := #MD_Timer.ET;
END_REGION

REGION Network 13: Calculate MD Frequence
   IF (#MD_Time_DINT > #MD_Time) OR #MD_Pulse THEN #MD_Time := #MD_Time_DINT; END_IF;
END_REGION

REGION Network 14: MD Timer
   // The MD_Timer is inserted twice to ensure that the timer is enabled in the same 
   // scan after af MD pulse.
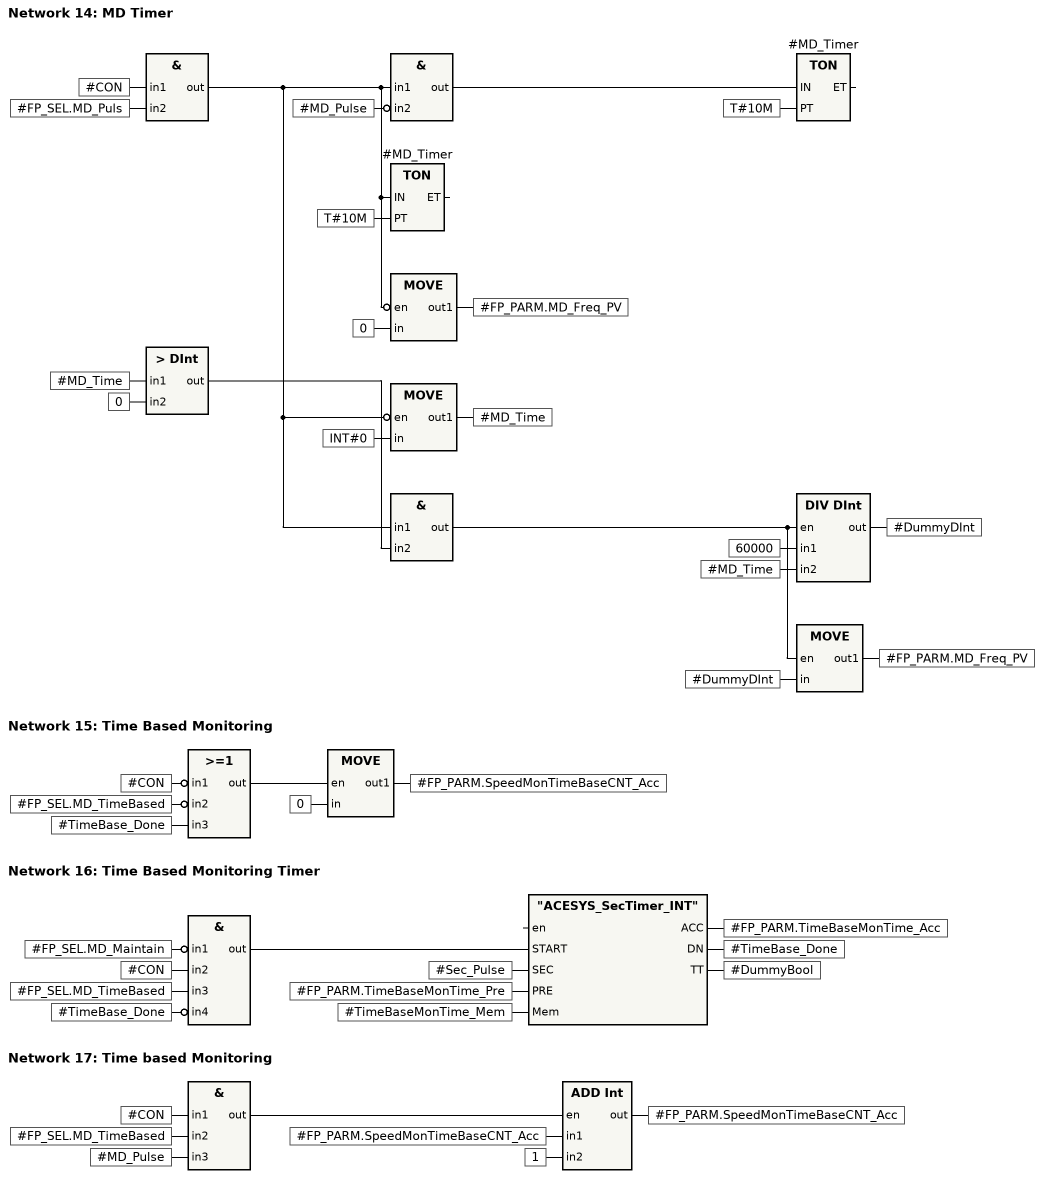
   #_w1 := #CON AND #FP_SEL.MD_Puls;
   #MD_Timer(IN := #_w1 AND NOT #MD_Pulse, PT := T#10M);   // TON
   #MD_Timer(IN := #_w1, PT := T#10M);   // TON
   IF NOT #_w1 THEN
       #FP_PARM.MD_Freq_PV := 0;
       #MD_Time := INT#0;
   END_IF;
   IF #_w1 AND (#MD_Time > 0) THEN
       #DummyDInt := 60000 / #MD_Time;
       #FP_PARM.MD_Freq_PV := #DummyDInt;
   END_IF;
END_REGION

REGION Network 15: Time Based Monitoring
   IF NOT #CON OR NOT #FP_SEL.MD_TimeBased OR #TimeBase_Done THEN
       #FP_PARM.SpeedMonTimeBaseCNT_Acc := 0;
   END_IF;
END_REGION

REGION Network 16: Time Based Monitoring Timer
   "ACESYS_SecTimer_INT"(START := NOT #FP_SEL.MD_Maintain AND #CON AND #FP_SEL.MD_TimeBased AND NOT #TimeBase_Done,
                         SEC := #Sec_Pulse,
                         PRE := #FP_PARM.TimeBaseMonTime_Pre,
                         Mem := #TimeBaseMonTime_Mem,
                         ACC => #FP_PARM.TimeBaseMonTime_Acc,
                         DN => #TimeBase_Done,
                         TT => #DummyBool);
END_REGION

REGION Network 17: Time based Monitoring
   IF #CON AND #FP_SEL.MD_TimeBased AND #MD_Pulse THEN
       #FP_PARM.SpeedMonTimeBaseCNT_Acc := #FP_PARM.SpeedMonTimeBaseCNT_Acc + 1;
   END_IF;
END_REGION

REGION Network 18: Time based Monitoring - Trig Alarm
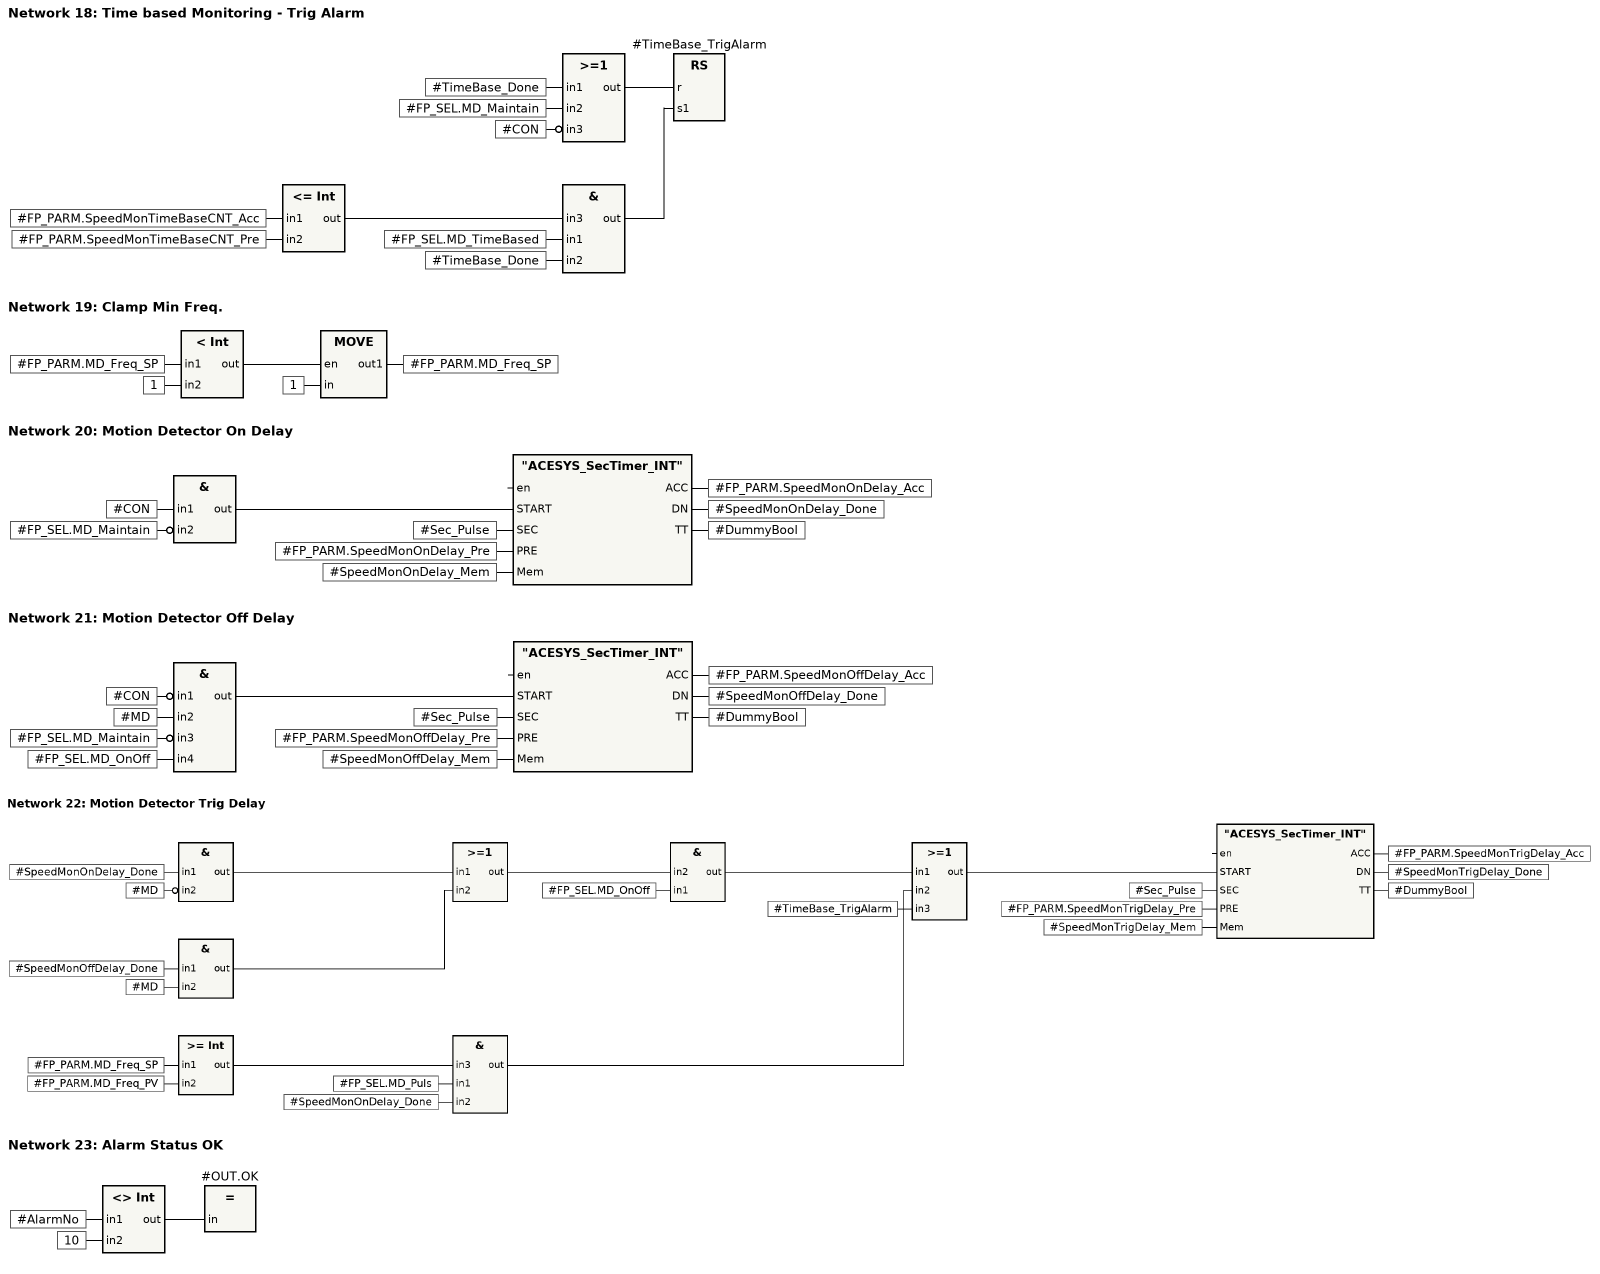
   IF #TimeBase_Done OR #FP_SEL.MD_Maintain OR NOT #CON THEN
       #TimeBase_TrigAlarm := FALSE;   // RS flip-flop
   END_IF;
   IF (#FP_PARM.SpeedMonTimeBaseCNT_Acc <= #FP_PARM.SpeedMonTimeBaseCNT_Pre) AND #FP_SEL.MD_TimeBased AND #TimeBase_Done THEN
       #TimeBase_TrigAlarm := TRUE;
   END_IF;
END_REGION

REGION Network 19: Clamp Min Freq.
   IF #FP_PARM.MD_Freq_SP < 1 THEN #FP_PARM.MD_Freq_SP := 1; END_IF;
END_REGION

REGION Network 20: Motion Detector On Delay
   "ACESYS_SecTimer_INT"(START := #CON AND NOT #FP_SEL.MD_Maintain,
                         SEC := #Sec_Pulse,
                         PRE := #FP_PARM.SpeedMonOnDelay_Pre,
                         Mem := #SpeedMonOnDelay_Mem,
                         ACC => #FP_PARM.SpeedMonOnDelay_Acc,
                         DN => #SpeedMonOnDelay_Done,
                         TT => #DummyBool);
END_REGION

REGION Network 21: Motion Detector Off Delay
   "ACESYS_SecTimer_INT"(START := NOT #CON AND #MD AND NOT #FP_SEL.MD_Maintain AND #FP_SEL.MD_OnOff,
                         SEC := #Sec_Pulse,
                         PRE := #FP_PARM.SpeedMonOffDelay_Pre,
                         Mem := #SpeedMonOffDelay_Mem,
                         ACC => #FP_PARM.SpeedMonOffDelay_Acc,
                         DN => #SpeedMonOffDelay_Done,
                         TT => #DummyBool);
END_REGION

REGION Network 22: Motion Detector Trig Delay
   "ACESYS_SecTimer_INT"(START := (((#SpeedMonOnDelay_Done AND NOT #MD) OR (#SpeedMonOffDelay_Done AND #MD)) AND #FP_SEL.MD_OnOff) OR ((#FP_PARM.MD_Freq_SP >= #FP_PARM.MD_Freq_PV) AND #FP_SEL.MD_Puls AND #SpeedMonOnDelay_Done) OR #TimeBase_TrigAlarm,
                         SEC := #Sec_Pulse,
                         PRE := #FP_PARM.SpeedMonTrigDelay_Pre,
                         Mem := #SpeedMonTrigDelay_Mem,
                         ACC => #FP_PARM.SpeedMonTrigDelay_Acc,
                         DN => #SpeedMonTrigDelay_Done,
                         TT => #DummyBool);
END_REGION

REGION Network 23: Alarm Status OK
   #OUT.OK := #AlarmNo <> 10;
END_REGION

REGION Network 24: Act as Dynamic sensor
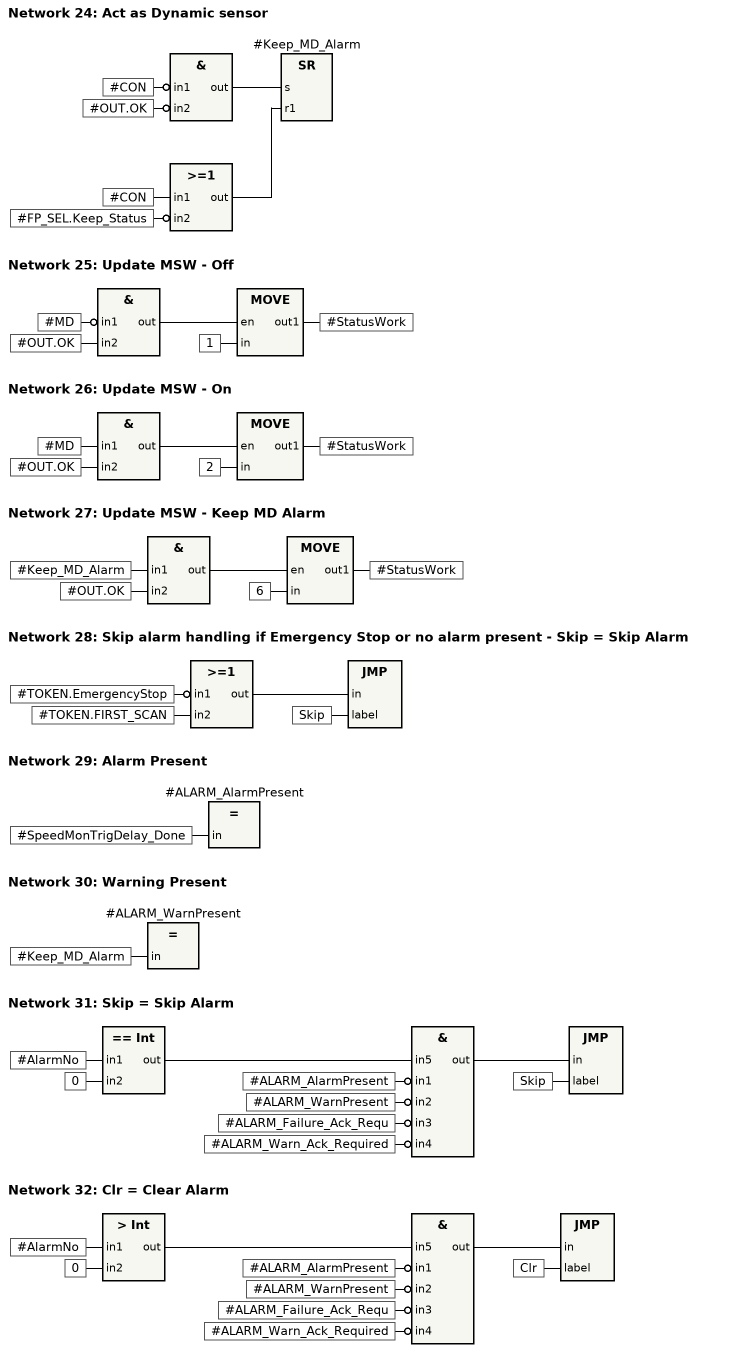
   IF NOT #CON AND NOT #OUT.OK THEN
       #Keep_MD_Alarm := TRUE;   // SR flip-flop
   END_IF;
   IF #CON OR NOT #FP_SEL.Keep_Status THEN #Keep_MD_Alarm := FALSE; END_IF;
END_REGION

REGION Network 25: Update MSW - Off
   IF NOT #MD AND #OUT.OK THEN #StatusWork := 1; END_IF;
END_REGION

REGION Network 26: Update MSW - On
   IF #MD AND #OUT.OK THEN #StatusWork := 2; END_IF;
END_REGION

REGION Network 27: Update MSW - Keep MD Alarm
   IF #Keep_MD_Alarm AND #OUT.OK THEN #StatusWork := 6; END_IF;
END_REGION

REGION Network 28: Skip alarm handling if Emergency Stop or no alarm present - Skip = Skip Alarm
   IF NOT #TOKEN.EmergencyStop OR #TOKEN.FIRST_SCAN THEN GOTO Skip; END_IF;
END_REGION

REGION Network 29: Alarm Present
   #ALARM_AlarmPresent := #SpeedMonTrigDelay_Done;
END_REGION

REGION Network 30: Warning Present
   #ALARM_WarnPresent := #Keep_MD_Alarm;
END_REGION

REGION Network 31: Skip = Skip Alarm
   IF (#AlarmNo = 0) AND NOT #ALARM_AlarmPresent AND NOT #ALARM_WarnPresent AND NOT #ALARM_Failure_Ack_Requ AND NOT #ALARM_Warn_Ack_Required THEN
       GOTO Skip;
   END_IF;
END_REGION

REGION Network 32: Clr = Clear Alarm
   IF (#AlarmNo > 0) AND NOT #ALARM_AlarmPresent AND NOT #ALARM_WarnPresent AND NOT #ALARM_Failure_Ack_Requ AND NOT #ALARM_Warn_Ack_Required THEN
       GOTO Clr;
   END_IF;
END_REGION

REGION Network 33: Ack = Alarm Acknowledge
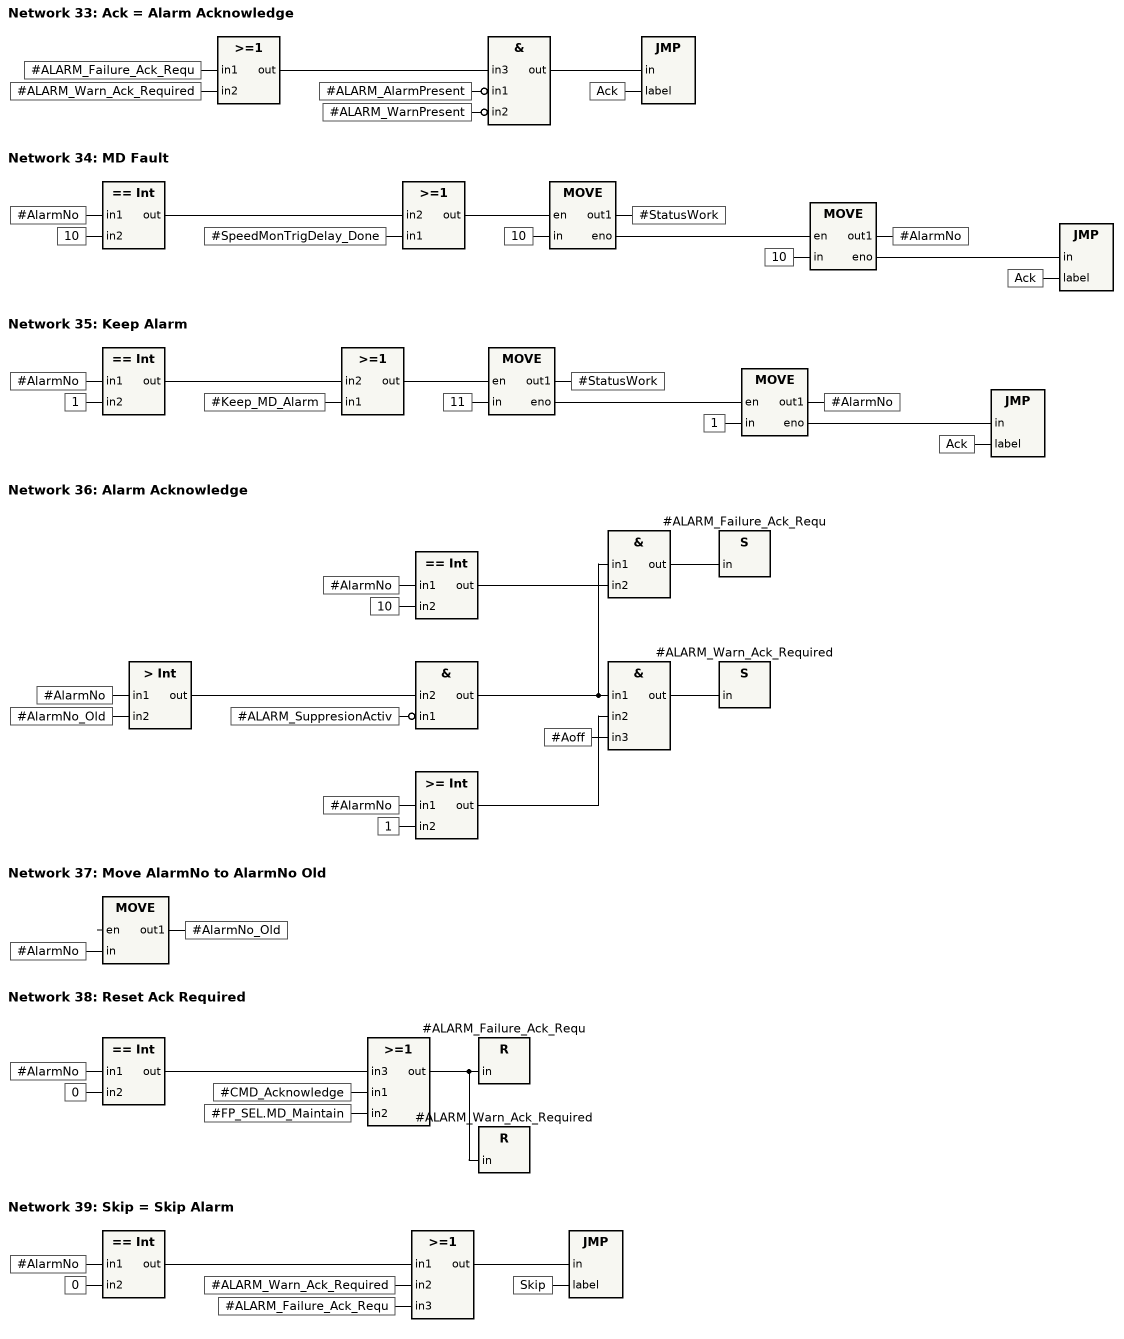
   IF (#ALARM_Failure_Ack_Requ OR #ALARM_Warn_Ack_Required) AND NOT #ALARM_AlarmPresent AND NOT #ALARM_WarnPresent THEN
       GOTO Ack;
   END_IF;
END_REGION

REGION Network 34: MD Fault
   // ENO of a box is taken as its EN; it also drops when the box reports an error
   #_w1 := (#AlarmNo = 10) OR #SpeedMonTrigDelay_Done;
   IF #_w1 THEN
       #StatusWork := 10;
       #AlarmNo := 10;
       GOTO Ack;
   END_IF;
END_REGION

REGION Network 35: Keep Alarm
   // ENO of a box is taken as its EN; it also drops when the box reports an error
   #_w1 := (#AlarmNo = 1) OR #Keep_MD_Alarm;
   IF #_w1 THEN
       #StatusWork := 11;
       #AlarmNo := 1;
       GOTO Ack;
   END_IF;
END_REGION

REGION Network 36: Alarm Acknowledge
   Ack:
   #_w1 := (#AlarmNo > #AlarmNo_Old) AND NOT #ALARM_SuppresionActiv;
   IF #_w1 AND (#AlarmNo = 10) THEN #ALARM_Failure_Ack_Requ := TRUE; END_IF;
   IF #_w1 AND (#AlarmNo >= 1) AND #Aoff THEN #ALARM_Warn_Ack_Required := TRUE; END_IF;
END_REGION

REGION Network 37: Move AlarmNo to AlarmNo Old
   #AlarmNo_Old := #AlarmNo;
END_REGION

REGION Network 38: Reset Ack Required
   IF (#AlarmNo = 0) OR #CMD_Acknowledge OR #FP_SEL.MD_Maintain THEN
       #ALARM_Failure_Ack_Requ := FALSE;
       #ALARM_Warn_Ack_Required := FALSE;
   END_IF;
END_REGION

REGION Network 39: Skip = Skip Alarm
   IF (#AlarmNo = 0) OR #ALARM_Warn_Ack_Required OR #ALARM_Failure_Ack_Requ THEN GOTO Skip; END_IF;
END_REGION

REGION Network 40: Clear Alarm - Label
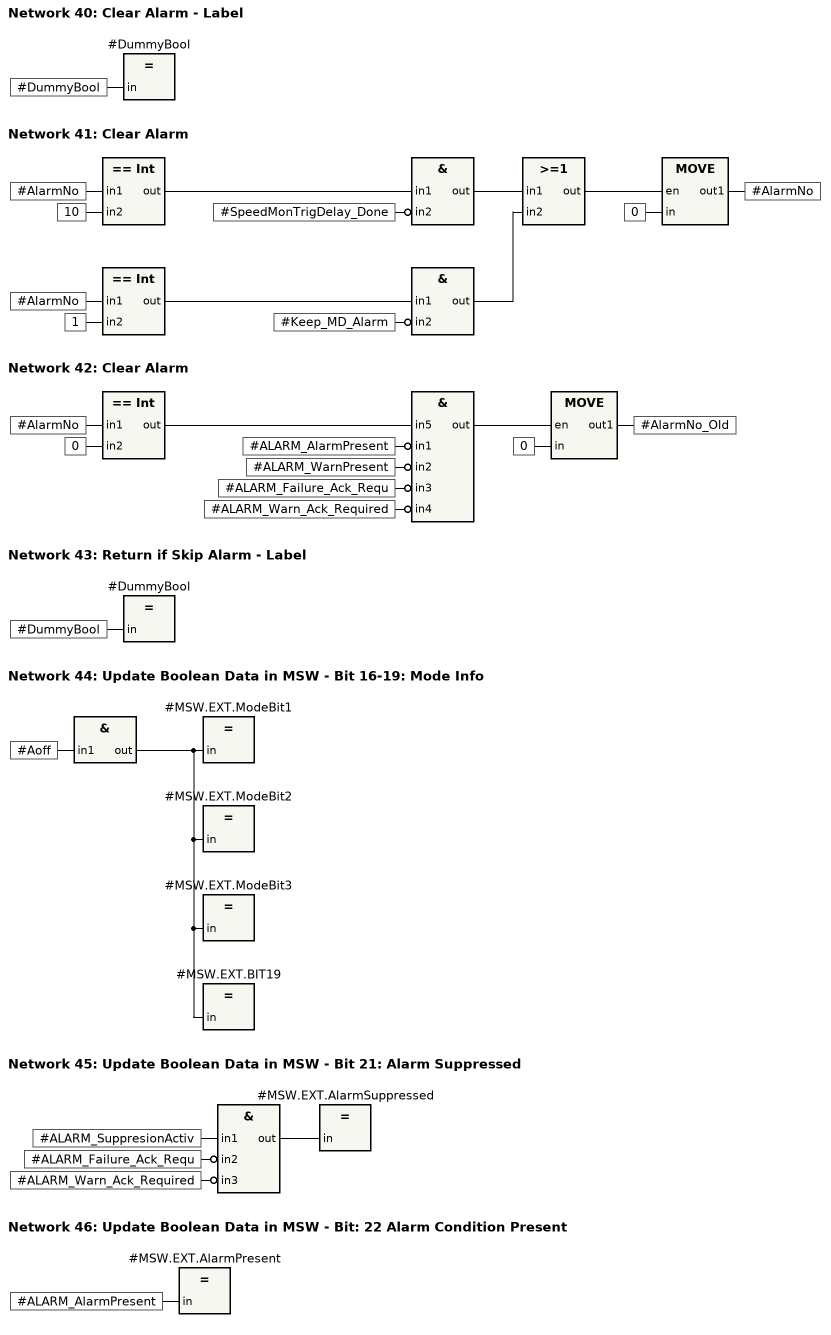
   Clr:
   #DummyBool := #DummyBool;
END_REGION

REGION Network 41: Clear Alarm
   IF ((#AlarmNo = 10) AND NOT #SpeedMonTrigDelay_Done) OR ((#AlarmNo = 1) AND NOT #Keep_MD_Alarm) THEN
       #AlarmNo := 0;
   END_IF;
END_REGION

REGION Network 42: Clear Alarm
   IF (#AlarmNo = 0) AND NOT #ALARM_AlarmPresent AND NOT #ALARM_WarnPresent AND NOT #ALARM_Failure_Ack_Requ AND NOT #ALARM_Warn_Ack_Required THEN
       #AlarmNo_Old := 0;
   END_IF;
END_REGION

REGION Network 43: Return if Skip Alarm - Label
   Skip:
   #DummyBool := #DummyBool;
END_REGION

REGION Network 44: Update Boolean Data in MSW - Bit 16-19: Mode Info
   // 0 = Auto
   // 1= Single Start
   // 2 = Manual
   // 3= Local
   // 4= Test Mode
   #MSW.EXT.ModeBit1 := #Aoff;
   #MSW.EXT.ModeBit2 := #Aoff;
   #MSW.EXT.ModeBit3 := #Aoff;
   #MSW.EXT.BIT19 := #Aoff;
END_REGION

REGION Network 45: Update Boolean Data in MSW - Bit 21: Alarm Suppressed
   #MSW.EXT.AlarmSuppressed := #ALARM_SuppresionActiv AND NOT #ALARM_Failure_Ack_Requ AND NOT #ALARM_Warn_Ack_Required;
END_REGION

REGION Network 46: Update Boolean Data in MSW - Bit: 22 Alarm Condition Present
   #MSW.EXT.AlarmPresent := #ALARM_AlarmPresent;
END_REGION

REGION Network 47: Update Boolean Data in MSW - Bit 23: Alarm Failure Present or Unacknowledged
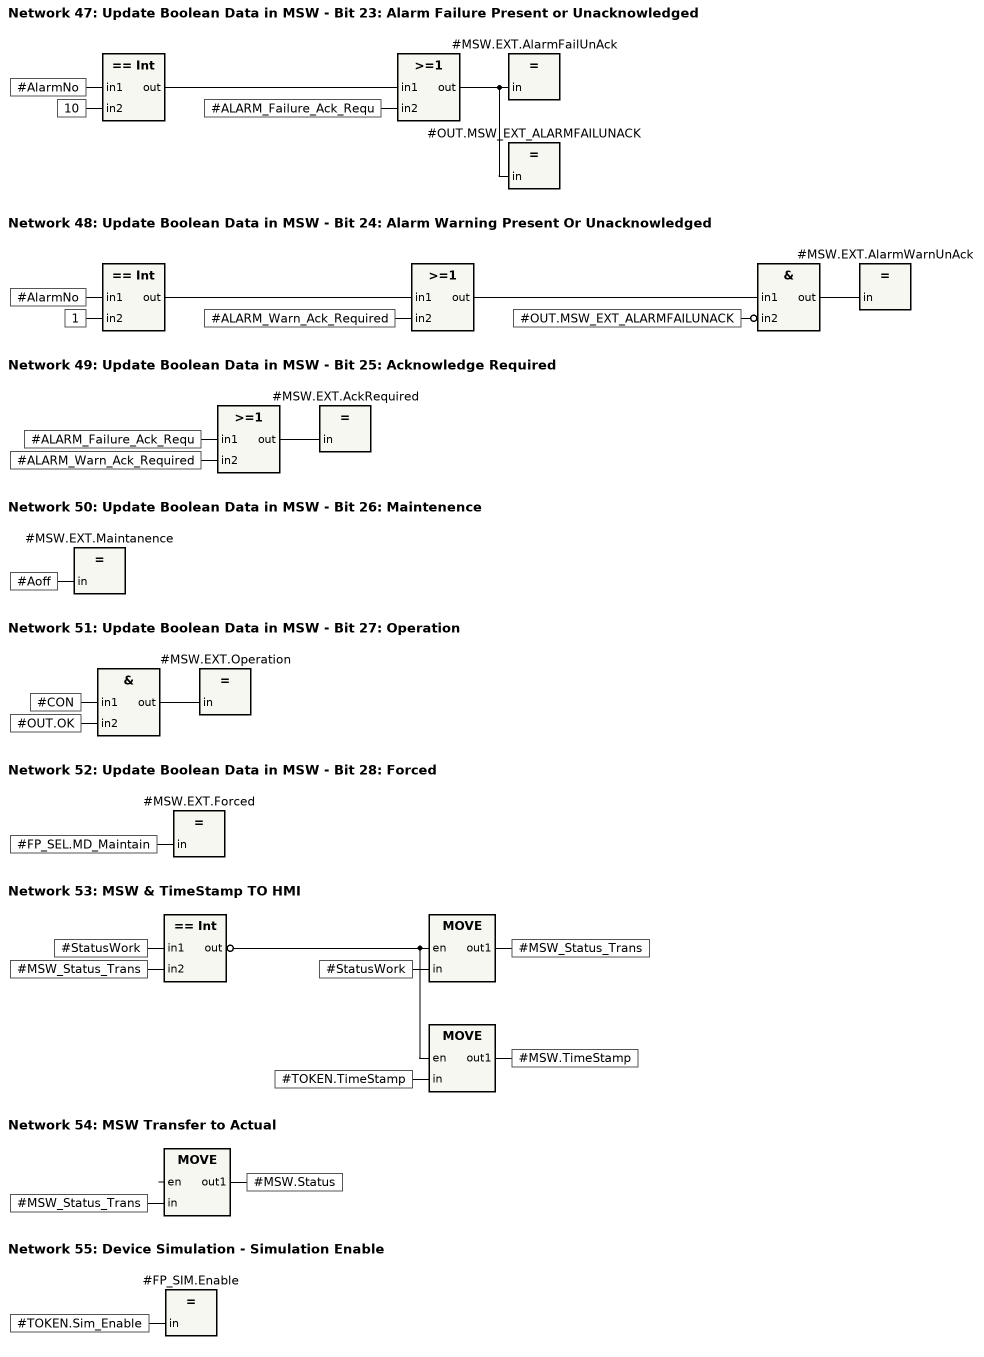
   #MSW.EXT.AlarmFailUnAck := (#AlarmNo = 10) OR #ALARM_Failure_Ack_Requ;
   #OUT.MSW_EXT_ALARMFAILUNACK := #MSW.EXT.AlarmFailUnAck;
END_REGION

REGION Network 48: Update Boolean Data in MSW - Bit 24: Alarm Warning Present Or Unacknowledged
   #MSW.EXT.AlarmWarnUnAck := ((#AlarmNo = 1) OR #ALARM_Warn_Ack_Required) AND NOT #OUT.MSW_EXT_ALARMFAILUNACK;
END_REGION

REGION Network 49: Update Boolean Data in MSW - Bit 25: Acknowledge Required
   #MSW.EXT.AckRequired := #ALARM_Failure_Ack_Requ OR #ALARM_Warn_Ack_Required;
END_REGION

REGION Network 50: Update Boolean Data in MSW - Bit 26: Maintenence
   #MSW.EXT.Maintanence := #Aoff;
END_REGION

REGION Network 51: Update Boolean Data in MSW - Bit 27: Operation
   #MSW.EXT.Operation := #CON AND #OUT.OK;
END_REGION

REGION Network 52: Update Boolean Data in MSW - Bit 28: Forced
   #MSW.EXT.Forced := #FP_SEL.MD_Maintain;
END_REGION

REGION Network 53: MSW & TimeStamp TO HMI
   #_w1 := NOT (#StatusWork = #MSW_Status_Trans);
   IF #_w1 THEN
       #MSW_Status_Trans := #StatusWork;
       #MSW.TimeStamp := #TOKEN.TimeStamp;
   END_IF;
END_REGION

REGION Network 54: MSW Transfer to Actual
   #MSW.Status := #MSW_Status_Trans;
END_REGION

REGION Network 55: Device Simulation - Simulation Enable
   #FP_SIM.Enable := #TOKEN.Sim_Enable;
END_REGION

REGION Network 56: Device Simulation - Seconds Pulse
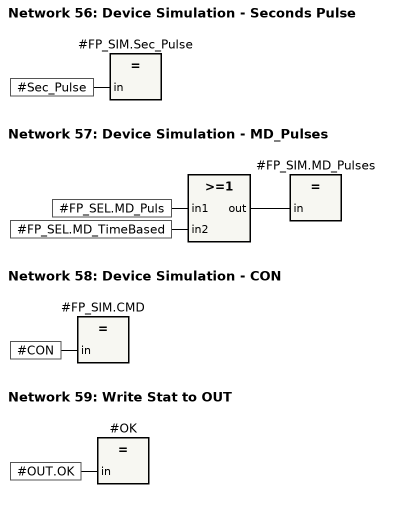
   #FP_SIM.Sec_Pulse := #Sec_Pulse;
END_REGION

REGION Network 57: Device Simulation - MD_Pulses
   #FP_SIM.MD_Pulses := #FP_SEL.MD_Puls OR #FP_SEL.MD_TimeBased;
END_REGION

REGION Network 58: Device Simulation - CON
   #FP_SIM.CMD := #CON;
END_REGION

REGION Network 59: Write Stat to OUT
   #OK := #OUT.OK;
END_REGION
END_FUNCTION_BLOCK

FUNCTION_BLOCK "ACESYS_MOTOR"   // FB210, FBD
TITLE = ACESYS V8.0 - Build 013 - MOTOR Block
{ S7_Optimized_Access := 'FALSE' }
AUTHOR : FLSmidth
FAMILY : ACESYS
NAME : MOTOR
VERSION : 8.0
   VAR_INPUT
      CMD : "ACESYS_GRP_CMD";
      SEL : Bool := TRUE;   // Unit Select by User program
      ASTR : Bool := TRUE;   // Auto Start
      DIR : Bool := TRUE;   // Direction ("1"=Direction 1 / "0"= Direction 2)
      MCC : Bool := TRUE;   // MCC Ready
      RDY : Bool := TRUE;   // Unit ready
      OVL : Bool := TRUE;   // Overload / trip
      RET1 : Bool;   // Feedback contactor 1
      RET2 : Bool;   // Feedback contactor 2
      LSTR1 : Bool;   // Local start 1
      LSTR2 : Bool;   // Local start 2
      LSTP : Bool := TRUE;   // Local stop
      REM : Bool := TRUE;   // Unit in Remote operation
      SSW : Bool := TRUE;   // Safety switch
      TFA : Bool := TRUE;   // Termistor fault
      DRDY : Bool := TRUE;   // Drive / MCC ready
      MD : Bool := TRUE;   // Motion detactor
      STALL : Bool := TRUE;   // Motor stalled
      EARTH : Bool := TRUE;   // Earth fault
      UBAL : Bool := TRUE;   // Unbalance / Phase lost
      GFA : Bool := TRUE;   // General fault
      GWA : Bool := TRUE;   // General waring
      BUSF : Bool := TRUE;   // Bus failure
      DOPR : Bool := TRUE;   // Drawer in operation position
      DTEST : Bool;   // Drawer in test position
      SFS : Bool := TRUE;   // Starter First step
      SLS : Bool;   // Starter in last step
      ES : Bool;   // Excessive starts
      ACK : Bool;   // Feedback from unit on alarm reset
      AI1 : Real;   // Analog value 1
      AI2 : Real;   // Analog value 2
      AI3 : Real;   // Analog value 3
      SPSET : Real;   // Speed setpoint
   END_VAR
   VAR_OUTPUT
      INTL : "ACESYS_INTL";   // Interlock
      INTL_SEQ_STR1 : "ACESYS_INTL";   // Interlock Sequence Start
      INTL_SEQ_STR2 : "ACESYS_INTL";   // Interlock Sequence Start
      INTL_SEQ_STP : "ACESYS_INTL";   // Interlock Sequence Stop
      CON1 : Bool;   // Command 1
      CON2 : Bool;   // Command 2
      LAMP1 : Bool;   // Lamp 1
      LAMP2 : Bool;   // Lamp 2
      SACK : Bool;   // Start Acknowledge
      RD1 : Bool;   // Run delayed 1
      RD2 : Bool;   // Run delayed 2
      RUN1 : Bool;   // Run 1
      RUN2 : Bool;   // Run 2
      OK : Bool;   // Unit Status OK (no alarms)
      LOC : Bool;   // Unit in Local Mode
      MAN : Bool;   // Unit in Manual Mode
      AUT : Bool;   // Unit in Auto Mode
      SS : Bool;   // Unit in Single Start Mode
      RES : Bool;   // Reset to unit
      TESTP : Bool;   // Test mode permission to unit
      ASTW : Bool;   // Start warning
      AL_SUPR : Bool;   // Supress Child Alarms
      AO1a : Real;   // Analog converted 1a
      AO1b : Real;   // Analog converted 1b
      AO2a : Real;   // Analog converted 2a
      AO2b : Real;   // Analog converted 2b
      AO3a : Real;   // Analog converted 3a
      AO3b : Real;   // Analog converted 3b
      CV : Real;   // Speed setpoint to VFD
      MSW : "ACESYS_HMI_STAT_32T";
   END_VAR
   VAR_IN_OUT
      TOKEN : "ACESYS_TOKEN";
   END_VAR
   VAR
      BlockInfo : Struct
         Ace_Version : Int;   // Acesys Block Version Number
         Ace_BuildNo : Int;   // Acesys Block Build Number
         State_Act : Int;   // Actual State Number
         State_Prev : Int;   // Previous State Number
         DB_Number : Int;   // Block Instance DB Number
      END_STRUCT;
      FP_CMD : Struct   // Faceplate Commands
         QuickStop : Bool;
         Spare_09 : Bool;
         Spare_10 : Bool;
         Spare_11 : Bool;
         Spare_12 : Bool;
         Spare_13 : Bool;
         Spare_14 : Bool;
         AckAlarm : Bool;
         Auto : Bool;
         Manual : Bool;
         Local : Bool;
         Start1 : Bool;
         Start2 : Bool;
         Stop : Bool;
         Reset : Bool;
         Test : Bool;
      END_STRUCT;
      FP_SEL : Struct   // Faceplate Selections
         MD : Bool;   // Motion Detector: Pulse Type
         MD_Puls : Bool;   // Motion Detector: Pulse Type
         MD_OnOff : Bool;   // Motion Detector: On/Off Type
         MD_Maintain : Bool;   // Faceplate Toggle MD Service
         STW_AutoStart : Bool;   // Faceplate Start Warning in Auto Start mode
         STW_Local : Bool;   // Faceplate Start Warning in Local mode
         STW_Manual : Bool;   // Faceplate Start Warning in Manual mode
         STW_Single : Bool;   // Faceplate Start Warning in Single Start mode
         Type_Unimotor : Bool;   // Faceplate Unimotor type
         Type_Bimotor : Bool;   // Faceplate Bimotor type
         Type_Indication : Bool;   // Faceplate Indication type
         MotorStarter : Bool;   // Faceplate Motor Starter Selected
         ParentSupress : Bool;   // Enable Parent Supress of alarms
         ParentCollection : Bool;   // Enable Inching in Manual Mode
         INCH_Man : Bool;   // Enable Inching in Manual Mode
         INCH_Loc : Bool;   // Enable Inching in Local Mode
         OutOfSevice : Bool;   // Select Out of Service
         WarningDrive : Bool;   // 0 = Failure Drive / 1 = Warning Drive
         Spare14 : Bool;
         Spare13 : Bool;
         Spare12 : Bool;
         Spare11 : Bool;
         Spare10 : Bool;
         Spare9 : Bool;
         Spare8 : Bool;
         Spare7 : Bool;
         Spare6 : Bool;
         Spare5 : Bool;
         Spare4 : Bool;
         Spare3 : Bool;
         Spare2 : Bool;
         Spare1 : Bool;
      END_STRUCT;
      FP_EN : Struct
         Mode_Auto : Bool;
         Mode_Man : Bool;
         Mode_Loc : Bool;
         Mode_Test : Bool;
         Mode_SS_Field : Bool;
         Mode_SS_FP : Bool;
         PB_QStop : Bool;
         Spare9 : Bool;
         Spare8 : Bool;
         Spare7 : Bool;
         Spare6 : Bool;
         Spare5 : Bool;
         Spare4 : Bool;
         Spare3 : Bool;
         Spare2 : Bool;
         Spare1 : Bool;
      END_STRUCT;
      FP_DIM : Struct   // Faceplate Dimmed Buttons
         Auto : Bool;
         Local : Bool;
         Manual : Bool;
         Start1 : Bool;
         Start2 : Bool;
         Stop : Bool;
         TEst : Bool;
         QStop : Bool;
         Reset : Bool;
         Spare7 : Bool;
         Spare6 : Bool;
         Spare5 : Bool;
         Spare4 : Bool;
         Spare3 : Bool;
         Spare2 : Bool;
         Spare1 : Bool;
      END_STRUCT;
      FP_SHOW : Struct   // Faceplate Show Buttons
         PB_Auto : Bool;
         PB_Local : Bool;
         PB_Manual : Bool;
         PB_Start1 : Bool;
         PB_Start2 : Bool;
         PB_Stop : Bool;
         PB_Test : Bool;
         PB_QStop : Bool;
         AI1 : Bool;
         AI2 : Bool;
         AI3 : Bool;
         SP : Bool;
         MCC : Bool;
         RDY : Bool;
         OVL : Bool;
         LSTP : Bool;
         REM : Bool;
         SSW : Bool;
         ES : Bool;
         TFA : Bool;
         DRDY : Bool;
         STALL : Bool;
         EARTH : Bool;
         UBAL : Bool;
         GFA : Bool;
         GWA : Bool;
         BUSF : Bool;
         DOPR : Bool;
         DTEST : Bool;
         ACK : Bool;
         LSTR1 : Bool;
         LSTR2 : Bool;
         RET2 : Bool;
         RUN2 : Bool;
         CON2 : Bool;
         RD2 : Bool;
         SFS : Bool;
         SLS : Bool;
         MD : Bool;
         DelayRun2 : Bool;
         ChangeDir : Bool;
         PB_Reset : Bool;
         ASTR : Bool;
         Spare05 : Bool;
         Spare04 : Bool;
         Spare03 : Bool;
         Spare02 : Bool;
         Spare01 : Bool;
      END_STRUCT;
      FP_PARM : Struct   // Faceplate Parameters
         StartWarn_Pre : Int;
         StartWarn_Acc : Int;
         RunDelay1_Pre : Int;
         RunDelay1_Acc : Int;
         RunDelay2_Pre : Int;
         RunDelay2_Acc : Int;
         DelayStart_Pre : Int;
         DelayStart_Acc : Int;
         DelayStop_Pre : Int;
         DelayStop_Acc : Int;
         ReturnMon_Pre : Int;
         ReturnMon_Acc : Int;
         SpeedMonOnDelay_Pre : Int;
         SpeedMonOnDelay_Acc : Int;
         SpeedMonOffDelay_Pre : Int;
         SpeedMonOffDelay_Acc : Int;
         SpeedMonTrigDelay_Pre : Int;
         SpeedMonTrigDelay_Acc : Int;
         ChangeDir_Pre : Int;
         ChangeDir_Acc : Int;
         LeaveFS_Pre : Int;
         LeaveFS_Acc : Int;
         ReachLS_Pre : Int;
         ReachLS_Acc : Int;
         ReachFS_Pre : Int;
         ReachFS_Acc : Int;
         MD_Freq_SP : Int;
         MD_Freq_PV : Int;
         StopReason : Int;
         AI1_Max : Real;
         AI1_Min : Real;
         AI2_Max : Real;
         AI2_Min : Real;
         AI3_Max : Real;
         AI3_Min : Real;
         AO1a_Max : Real;
         AO1a_Min : Real;
         AO2a_Max : Real;
         AO2a_Min : Real;
         AO3a_Max : Real;
         AO3a_Min : Real;
         AO1b_Max : Real;
         AO1b_Min : Real;
         AO2b_Max : Real;
         AO2b_Min : Real;
         AO3b_Max : Real;
         AO3b_Min : Real;
         INTL : Bool;   // Interlock
         INTL_SEQ_STR1 : Bool;   // Interlock Sequence Start
         INTL_SEQ_STR2 : Bool;   // Interlock Sequence Start
         INTL_SEQ_STP : Bool;   // Interlock Sequence Stop
         Spare12 : Bool;
         Spare11 : Bool;
         Spare10 : Bool;
         Spare09 : Bool;
         Spare08 : Bool;
         Spare07 : Bool;
         Spare06 : Bool;
         Spare05 : Bool;
         Spare04 : Bool;
         Spare03 : Bool;
         Spare02 : Bool;
         Spare01 : Bool;
      END_STRUCT;
      FP_SIM : "ACESYS_SIM_MOTOR";
      AdapterBlock : "ACESYS_ADPT_MOTOR";
      STATE : Struct
         A_AutoStart1 : Bool;
         A_AutoStart2 : Bool;
         A_DelayedStart1 : Bool;
         A_DelayedStart2 : Bool;
         A_DelayedStop1 : Bool;
         A_DelayedStop2 : Bool;
         A_Running1 : Bool;
         A_Running2 : Bool;
         A_Selected1 : Bool;
         A_Selected2 : Bool;
         A_SelToStop1 : Bool;
         A_SelToStop2 : Bool;
         A_Stopping1 : Bool;
         A_Stopping2 : Bool;
         A_SeqStart1 : Bool;
         A_SeqStart2 : Bool;
         A_SeqStop1 : Bool;
         A_SeqStop2 : Bool;
         A_Starting1 : Bool;
         A_Starting2 : Bool;
         A_StartWarning1 : Bool;
         A_StartWarning2 : Bool;
         A_Stopped1 : Bool;
         A_Stopped2 : Bool;
         S_AutoStart1 : Bool;
         S_AutoStart2 : Bool;
         S_Running1 : Bool;
         S_Running2 : Bool;
         S_Starting1 : Bool;
         S_Starting2 : Bool;
         S_StartWarning1 : Bool;
         S_StartWarning2 : Bool;
         S_Stopped1 : Bool;
         S_Stopped2 : Bool;
         M_Running1 : Bool;
         M_Running2 : Bool;
         M_Starting1 : Bool;
         M_Starting2 : Bool;
         M_StartWarning1 : Bool;
         M_StartWarning2 : Bool;
         M_Stopped : Bool;
         L_Running1 : Bool;
         L_Running2 : Bool;
         L_Starting1 : Bool;
         L_Starting2 : Bool;
         L_StartWarning1 : Bool;
         L_StartWarning2 : Bool;
         L_Stopped : Bool;
         T_Starting1 : Bool;
         T_Starting2 : Bool;
         T_TestMode : Bool;
         T_TestPermission : Bool;
         Alarm : Bool;
         Interlock : Bool;
         EmergencyStop : Bool;
         OutOfService : Bool;
      END_STRUCT;
      ONS : Struct
         Unimotor : Bool;
         Bimotor : Bool;
         MD_OnOff : Bool;
         MD_Puls : Bool;
         LSTR1_1 : Bool;
         LSTR1_2 : Bool;
         LSTR2_1 : Bool;
         LSTR2_2 : Bool;
         AckAlarm : Bool;
         Cmd_Auto : Bool;
         Cmd_Manual : Bool;
         CMD_Local : Bool;
         CMD_Test : Bool;
         GLTP : Bool;
         RET1 : Bool;
         RET2 : Bool;
         MD_Pulse : Bool;
         CMD_Start1 : Bool;
         CMD_Start2 : Bool;
         FP_Start1_CMD : Bool;
         FP_Start2_CMD : Bool;
         SecPulse1 : Bool;
         SecPulse2 : Bool;
         GSS_On : Bool;
         Spare8 : Bool;
         Spare7 : Bool;
         Spare6 : Bool;
         Spare5 : Bool;
         Spare4 : Bool;
         Spare3 : Bool;
         Spare2 : Bool;
         Spare1 : Bool;
      END_STRUCT;
      StatusWork : Int;
      ModePointer : Int;
      AlarmNo : Int;
      AlarmNo_Old : Int;
      StartWarn_Mem : Int;
      RunDelay1_Mem : Int;
      RunDelay2_Mem : Int;
      DelayStart_Mem : Int;
      DelayStop_Mem : Int;
      ReturnMon_Mem : Int;
      SpeedMonOnDelay_Mem : Int;
      SpeedMonOffDelay_Mem : Int;
      SpeedMonTrigDelay_Mem : Int;
      ChangeDir1_Mem : Int;
      ChangeDir2_Mem : Int;
      LeaveFS_Mem : Int;
      ReachLS_Mem : Int;
      ReachFS_Mem : Int;
      MD_Time : DInt;
      MD_Time_DINT : DInt;
      MD_Timer : TON_TIME;
      ModeAuto : Bool;
      ModeLocal : Bool;
      ModeManual : Bool;
      ModeSingleStart : Bool;
      ModeTest : Bool;
      Select : Bool;   // Parent & Program Select
      CMD_AckAlarm : Bool;
      CMD_Start1 : Bool;
      CMD_Start2 : Bool;
      CMD_Stop : Bool;
      CMD_QStop : Bool;
      CMD_Reset : Bool;
      FromStateAuto : Bool;
      FromStateSingle : Bool;
      FromStateManual : Bool;
      FromStateLocal : Bool;
      FromStateTest : Bool;
      FromStopState : Bool;
      ALARM_SupressionActive : Bool;
      ALARM_AlarmPresent : Bool;
      ALARM_WarnPresent : Bool;
      ALARM_FailureAckRequired : Bool;
      ALARM_WarnAckRequired : Bool;
      StartWarn_TT : Bool;
      StartWarn_Done : Bool;
      Rundelay1_Done : Bool;
      Rundelay2_Done : Bool;
      DelayStart_Done : Bool;
      DelayStop_Done : Bool;
      ReturnMon_Done : Bool;
      SpeedMonOnDelay_Done : Bool;
      SpeedMonOffDelay_Done : Bool;
      SpeedMonTrigDelay_Done : Bool;
      ChangeDir1_Done : Bool;
      ChangeDir2_Done : Bool;
      ChangeDir1_TT : Bool;
      ChangeDir2_TT : Bool;
      LeaveFS_Done : Bool;
      ReachLS_Done : Bool;
      ReachFS_Done : Bool;
      Trig_RET_ALARM : Bool;
      Trig_MD_ALARM : Bool;
      Trig_SFSNotLeave : Bool;
      Trig_SLSNotReach : Bool;
      Trig_SFSNotReach : Bool;
      Trig_SFSandSLS : Bool;
      RET1_OneScan : Bool;
      RET2_OneScan : Bool;
      MD_Pulse : Bool;
      NotEmpty : Bool;   // Unit Stopped un-normal
      LSTR1_Puls : Bool;
      LSTR2_Puls : Bool;
      Sec_Pulse : Bool;
      OUT : Struct
         CON1 : Bool;
         CON2 : Bool;
         LAMP1 : Bool;
         LAMP2 : Bool;
         SACK : Bool;
         RD1 : Bool;
         RD2 : Bool;
         RUN1 : Bool;
         RUN2 : Bool;
         OK : Bool;
         LOC : Bool;
         MAN : Bool;
         AUT : Bool;
         SS : Bool;
         RES : Bool;
         TESTP : Bool;
         ASTW : Bool;
         AL_SUPR : Bool;
         INTL_OK_STAT : Bool;
         INTL_SEQ_STR1_OK_STAT : Bool;
         INTL_SEQ_STR2_OK_STAT : Bool;
         INTL_SEQ_STP_OK_STAT : Bool;
      END_STRUCT;
      MSW_Status_Trans : Int;
   END_VAR
   VAR_TEMP
      AOn : Bool;   // Always On
      AOff : Bool;   // Always Off
      DummyBool : Bool;
      Temp_CON1 : Bool;
      Temp_CON2 : Bool;
      StatPointer_Old : Int;
      ChangeDir1_Acc : Int;
      ChangeDir2_Acc : Int;
      StatusBuilder : Int;
      DummyDINT : DInt;
      Status_Add : Int;
      DIR_Temp : Bool;
      RET2_Temp : Bool;
      LSTR2_Temp : Bool;
   END_VAR
   VAR_TEMP   // added for the SCL form of the ladder/FBD networks
      _w1 : Bool;
      _w2 : Bool;
      _w3 : Bool;
      _w4 : Bool;
      _w5 : Bool;
      _w6 : Bool;
      _w7 : Bool;
      _w8 : Bool;
   END_VAR
BEGIN

REGION Network 1: Always On
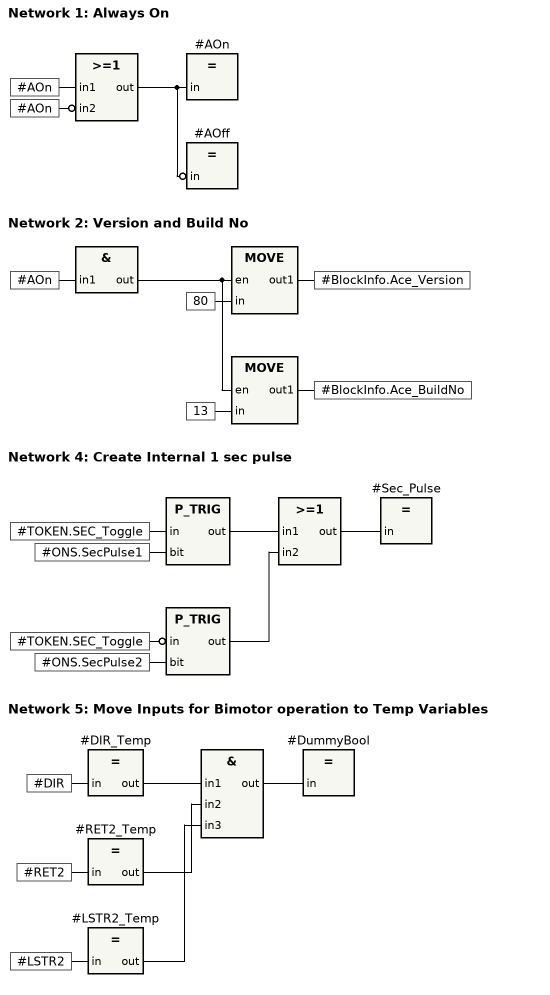
   #AOn := #AOn OR NOT #AOn;
   #AOff := NOT #AOn;
END_REGION

REGION Network 2: Version and Build No
   IF #AOn THEN
       #BlockInfo.Ace_Version := 80;
       #BlockInfo.Ace_BuildNo := 13;
   END_IF;
END_REGION

REGION Network 3 (STL): Instance DB Number to Faceplate
         L     DINO;
         T     #BlockInfo.DB_Number;
END_REGION

REGION Network 4: Create Internal 1 sec pulse
   #_w1 := #TOKEN.SEC_Toggle AND NOT #ONS.SecPulse1;   // rising edge
   #ONS.SecPulse1 := #TOKEN.SEC_Toggle;
   #_w2 := NOT #TOKEN.SEC_Toggle AND NOT #ONS.SecPulse2;   // rising edge
   #ONS.SecPulse2 := NOT #TOKEN.SEC_Toggle;
   #Sec_Pulse := #_w1 OR #_w2;
END_REGION

REGION Network 5: Move Inputs for Bimotor operation to Temp Variables
   #DIR_Temp := #DIR;
   #RET2_Temp := #RET2;
   #LSTR2_Temp := #LSTR2;
   #DummyBool := #DIR AND #RET2 AND #LSTR2;
END_REGION

REGION Network 6: Type Select
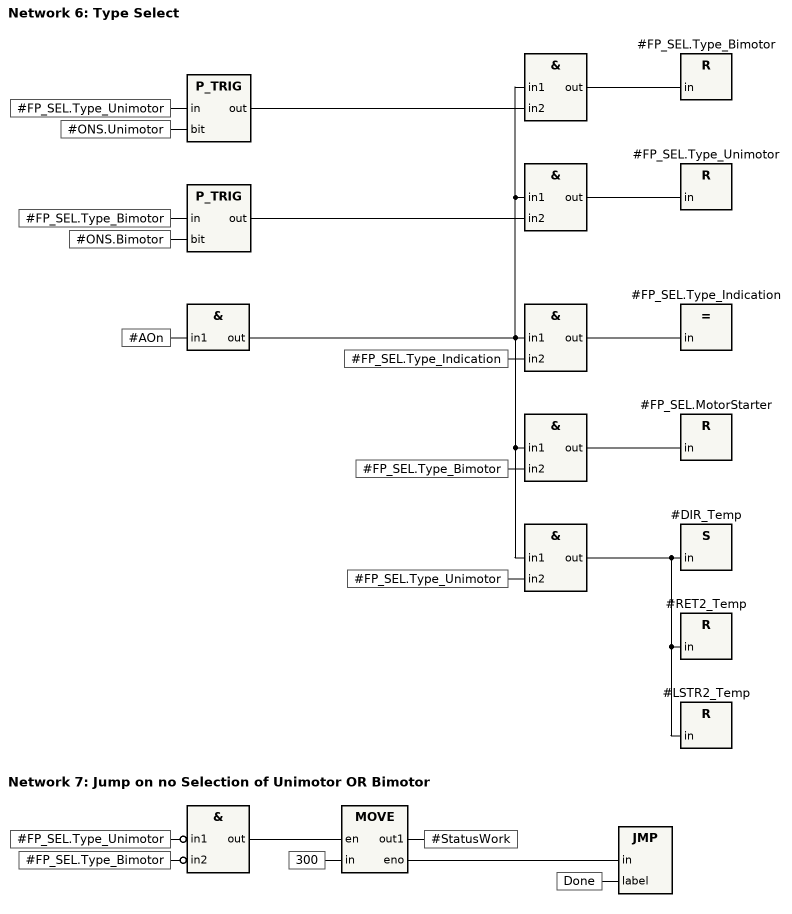
   #_w1 := #FP_SEL.Type_Unimotor AND NOT #ONS.Unimotor;   // rising edge
   #ONS.Unimotor := #FP_SEL.Type_Unimotor;
   IF #AOn AND #_w1 THEN #FP_SEL.Type_Bimotor := FALSE; END_IF;
   #_w2 := #FP_SEL.Type_Bimotor AND NOT #ONS.Bimotor;   // rising edge
   #ONS.Bimotor := #FP_SEL.Type_Bimotor;
   IF #AOn AND #_w2 THEN #FP_SEL.Type_Unimotor := FALSE; END_IF;
   #FP_SEL.Type_Indication := #AOn AND #FP_SEL.Type_Indication;
   IF #AOn AND #FP_SEL.Type_Bimotor THEN #FP_SEL.MotorStarter := FALSE; END_IF;
   IF #AOn AND #FP_SEL.Type_Unimotor THEN
       #DIR_Temp := TRUE;
       #RET2_Temp := FALSE;
       #LSTR2_Temp := FALSE;
   END_IF;
END_REGION

REGION Network 7: Jump on no Selection of Unimotor OR Bimotor
   // ENO of a box is taken as its EN; it also drops when the box reports an error
   #_w1 := NOT #FP_SEL.Type_Unimotor AND NOT #FP_SEL.Type_Bimotor;
   IF #_w1 THEN
       #StatusWork := 300;
       GOTO Done;
   END_IF;
END_REGION

REGION Network 8: Motion Detector
   // Build 007 - 03. Dec 2019 (EXTBOB) : Sel_MD_Maintain set to 0 when motion detector selection is deselected
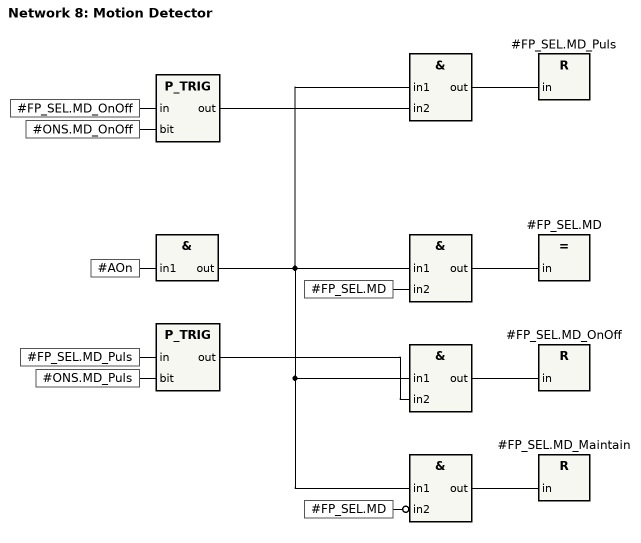
   #FP_SEL.MD := #AOn AND #FP_SEL.MD;
   #_w1 := #FP_SEL.MD_OnOff AND NOT #ONS.MD_OnOff;   // rising edge
   #ONS.MD_OnOff := #FP_SEL.MD_OnOff;
   IF #AOn AND #_w1 THEN #FP_SEL.MD_Puls := FALSE; END_IF;
   #_w2 := #FP_SEL.MD_Puls AND NOT #ONS.MD_Puls;   // rising edge
   #ONS.MD_Puls := #FP_SEL.MD_Puls;
   IF #AOn AND #_w2 THEN #FP_SEL.MD_OnOff := FALSE; END_IF;
   IF #AOn AND NOT #FP_SEL.MD THEN #FP_SEL.MD_Maintain := FALSE; END_IF;
END_REGION

REGION Network 9 (SCL): Transfer Interlock OK to Stat
   #OUT.INTL_OK_STAT := PEEK_BOOL(area := 16#84, dbNumber := #BlockInfo.DB_Number, byteOffset := 22, bitOffset := 0);
   #OUT.INTL_SEQ_STR1_OK_STAT := PEEK_BOOL(area := 16#84, dbNumber := #BlockInfo.DB_Number, byteOffset := 24, bitOffset := 0);
   #OUT.INTL_SEQ_STR2_OK_STAT := PEEK_BOOL(area := 16#84, dbNumber := #BlockInfo.DB_Number, byteOffset := 26, bitOffset := 0);
   #OUT.INTL_SEQ_STP_OK_STAT := PEEK_BOOL(area := 16#84, dbNumber := #BlockInfo.DB_Number, byteOffset := 28, bitOffset := 0);
END_REGION

REGION Network 10: Set Show Parameters
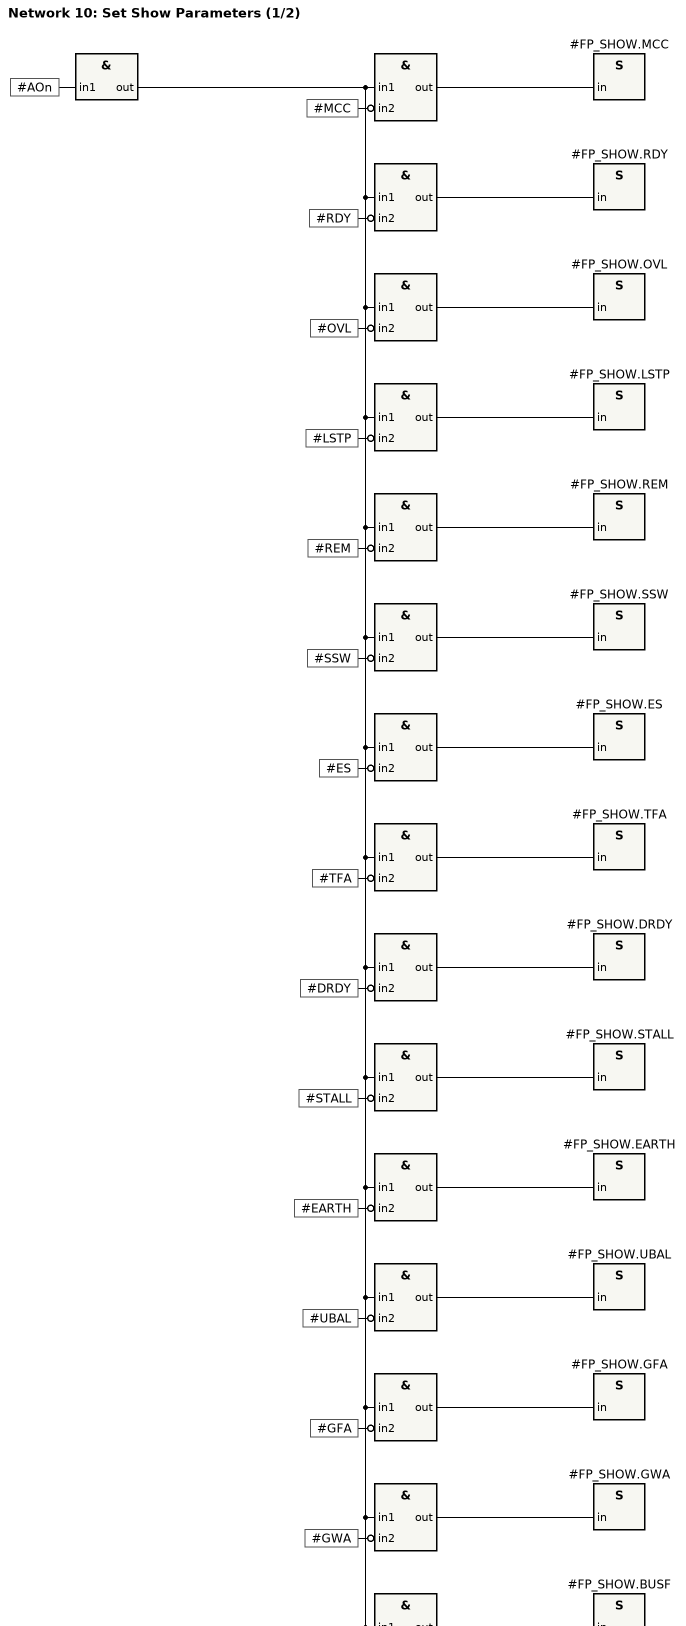
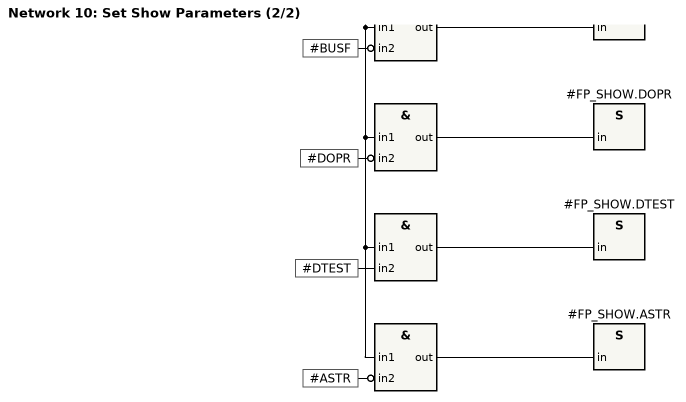
   IF #AOn AND NOT #MCC THEN #FP_SHOW.MCC := TRUE; END_IF;
   IF #AOn AND NOT #RDY THEN #FP_SHOW.RDY := TRUE; END_IF;
   IF #AOn AND NOT #OVL THEN #FP_SHOW.OVL := TRUE; END_IF;
   IF #AOn AND NOT #LSTP THEN #FP_SHOW.LSTP := TRUE; END_IF;
   IF #AOn AND NOT #REM THEN #FP_SHOW.REM := TRUE; END_IF;
   IF #AOn AND NOT #SSW THEN #FP_SHOW.SSW := TRUE; END_IF;
   IF #AOn AND NOT #ES THEN #FP_SHOW.ES := TRUE; END_IF;
   IF #AOn AND NOT #TFA THEN #FP_SHOW.TFA := TRUE; END_IF;
   IF #AOn AND NOT #DRDY THEN #FP_SHOW.DRDY := TRUE; END_IF;
   IF #AOn AND NOT #STALL THEN #FP_SHOW.STALL := TRUE; END_IF;
   IF #AOn AND NOT #EARTH THEN #FP_SHOW.EARTH := TRUE; END_IF;
   IF #AOn AND NOT #UBAL THEN #FP_SHOW.UBAL := TRUE; END_IF;
   IF #AOn AND NOT #GFA THEN #FP_SHOW.GFA := TRUE; END_IF;
   IF #AOn AND NOT #GWA THEN #FP_SHOW.GWA := TRUE; END_IF;
   IF #AOn AND NOT #BUSF THEN #FP_SHOW.BUSF := TRUE; END_IF;
   IF #AOn AND NOT #DOPR THEN #FP_SHOW.DOPR := TRUE; END_IF;
   IF #AOn AND #DTEST THEN #FP_SHOW.DTEST := TRUE; END_IF;
   IF #AOn AND NOT #ASTR THEN #FP_SHOW.ASTR := TRUE; END_IF;
END_REGION

REGION Network 11: Set Show Parameters
   // Build 002 - 25 March 2019 - En_Mode_SS_Field flag added in LSTR1/2
